(* CODESYS project CoDeSyS_library_v0.4.0.0.library
   LanguageModelAttribute: qualified-access-only
   Author: Razumovskii
   Version: 0.4.0.0
   Description: Standart library for main typical devices
   Title: mt
   Company: MechaTronics

Project tree, tasks and I/O mapping:
  libraries: Standard, 3.5.18.0 (System); Util, 3.5.19.0 (System); CAA File, 3.5.19.0 (CAA Technical Workgroup); CmpApp, 3.5.17.0 (System); SysTypes Interfaces, * (System)
  global variables sys
  System/
    program pou99_End [ST]: sysLoadZero, sysDevListReset, sysDevListCheck
    Library UDTs/
      data type udtDTL
      data type udtTimer
      data type timerSec
      data type timerRtc
      data type udtCMD
      data type timerCnt
      data type udtDevAnalog
      data type udtState
      data type udtDevDiscrete
      function devAtoD [ST]
      function devDtoA [ST]
      data type udtNetDataDiscrete
      data type udtNetDataAnalog
      data type uniSwap
    Library Methods/
      function GetLibVersion [ST]
      function block DrvBase [ST]: scale, conv, alm, almS, ot, exe, inc, blink, switch
      function block DrvTimer [ST]: sec, cnt, rtc
      function mbSwap [ST]
    program pou00_Start [ST]: pulse, clock, dtl, pulseOne
    Library Lists/
      data type listDev
      data type listRange
      data type listDevLoad
    function block DrvRetain [ST]: custom, system
  Drivers/
    Devices/
      02. Discrete Output/
        data type cfgDO
        data type cfgDOA
        function block DrvDO [ST]: s12_state, s15_globalData, s00_globalCommands, s05_exe, s09_options, s18_netData
        data type udtCfgDO
        function block DrvDOA [ST]: s12_state, s00_globalCommands, s01_externalCommand, s05_exe, s06_delays, s16_timers, s15_globalData, s07_turnON, s08_turnOFF, s09_options
      06. Valve Discrete/
        data type cfgV
        data type stateV
        function block DrvV [ST]: s00_globalCommands, s01_externalCommand, s04_alarmsRaw, s05_exe, s06_delays, s07_turnON, s08_turnOFF, s09_options, s10_alarms, s11_reset, s12_state, s14_opTime, s15_globalData, s16_timers, s17_hmi, s20_test, s18_netData
        data type udtCfgV
        data type udtAlarmV
        function block SubCalibration [ST]
      01. Discrete Input/
        data type cfgDI
        function block DrvDI [ST]: s00_globalCommands, s12_state, s02_workMode, s03_filter, s05_exe, s16_timers, s15_globalData, s09_options, s18_netData
        data type udtCfgDI
      05. Motor Direct/
        data type cfgM
        data type stateM
        function block DrvM [ST]: s16_timers, s15_globalData, s12_state, s00_globalCommands, s06_delays, s05_exe, s01_externalCommand, s09_options, s08_turnOFF, s07_turnON, s11_reset, s04_alarmsRaw, s10_alarms, s17_hmi, s14_opTime, s20_test, s18_netData
        data type udtCfgM
        data type udtAlarmM
      04. Analog Output/
        SlowMode/
          function block SubFilter [ST]
          function block SubSlow [ST]
          data type udtCfgSlow
          data type cfgSlow
        data type udtCfgAO
        data type cfgAO
        function block DrvAO [ST]: s12_state, s17_hmi, s15_globalData, s00_globalCommands, s01_externalCommand, s05_exe, s09_options, s18_netData
        data type stateAO
        function block DrvAO_MV210 [ST]: s12_state, s17_hmi, s15_globalData, s00_globalCommands, s01_externalCommand, s05_exe, s09_options, s04_alarmsRaw, s11_reset, s18_netData
        MV210/
          data type udtAO_MV210_502
          data type udtAlarmAO_MV210
          data type stateAO_MV210
      03. Analog Input/
        data type listAISp
        data type cfgAI
        data type stateAI
        data type udtAlarmAI
        data type udtCfgAI
        function block DrvAI [ST]: s07_turnON, s17_hmi, s04_alarmsRaw, s00_globalCommands, s10_alarms, s11_reset, s16_timers, s15_globalData, s02_workMode, s03_filter, s05_exe, s06_delays, s08_turnOFF, s09_options, s12_state, s18_netData
        function block DrvAI_MV210 [ST]: s07_turnON, s17_hmi, s04_alarmsRaw, s00_globalCommands, s10_alarms, s11_reset, s16_timers, s15_globalData, s02_workMode, s03_filter, s05_exe, s06_delays, s08_turnOFF, s09_options, s12_state, s18_netData
        MV210/
          data type udtAI_MV210_101
          data type udtAlarmAI_MV210
          data type stateAI_MV210
      20. PID/
        data type udtCfgPID
        data type cfgPID
        function block DrvPID [ST]: s07_turnON, s06_delays, s05_exe, s03_filter, s00_globalCommands, s09_options, s11_reset, s12_state, s15_globalData, s17_hmi, s13_commands
        data type statePID
        data type udtAlarmPID
      10. Flowmeter/
        function block DrvFlow [ST]: s00_globalCommands, s05_exe, s09_options, s11_reset, s12_state, s15_globalData, s16_timers, s17_hmi, s02_workMode, s03_filter, s18_netData
        data type udtCfgFlow
        data type cfgFlow
        data type stateFlow
    Special/
      function block DrvStatistics [ST]: calcD, addValue, reset, resetList, calcA, calcMulti
      data type listStatistic
      data type cfgStatistic
*)

// System/Library UDTs/udtDTL
TYPE udtDTL :
STRUCT
	//Data Time List
		year			:UINT;
		month			:UINT;
		day				:UINT;
		hour			:UINT;
		minute			:UINT;
		second			:UINT;
		millisecond		:UINT;
		weekDay			:WEEKDAY;
END_STRUCT
END_TYPE

// System/Library UDTs/udtTimer
TYPE udtTimer :
STRUCT
	//configuration word for Timers
		start		:BOOL;			// 0:	starting command
		Q			:BOOL;			// 1:	Quit
		pause		:BOOL;			// 2:	Pause
		reset		:BOOL;			// 3:	reset actual point to zero
		SFC			:BOOL;			// 4:	signal front control
		//you add more configuration bits for the project, if necessary, but not more than 16
END_STRUCT
END_TYPE

// System/Library UDTs/timerSec
TYPE timerSec :
STRUCT
	//control struct for a Timer Second
		cmd			:udtTimer;		//command word
		sp			:INT := 2;		//set point
		ap			:INT;			//actual point	
END_STRUCT
END_TYPE

// System/Library UDTs/timerRtc
TYPE timerRtc :
STRUCT
	//control struct for a Timer High Accucary
		cmd			:udtTimer;		//command word
		sp			:REAL := 2.000;	//set point as second
		ap			:REAL;			//actual point	
		RTC			:UDINT;			//real time stamp
		delta		:UDINT;			//delta time control
		percent		:REAL;			//progress 0..100%
END_STRUCT
END_TYPE

// System/Library UDTs/udtCMD
TYPE udtCMD :
STRUCT
	//standart control word
		startA	 		:BOOL;		// 0:	command for automatic control
		startM	 		:BOOL;		// 1:	command for manual control
		manual			:BOOL;		// 2:	mode of control (0 - automatic, 1 - manual (user or HMI))
		lock			:BOOL;		// 3:	technological lock
		force			:BOOL;		// 4:	forced control in manual mode
		service			:BOOL;		// 5:	activate service mode
		local			:BOOL;		// 6: 	activate local mode (0 - controlled by PLC, 1 - controlled by local keys)
		reset			:BOOL;		// 7:	resetting of device
		alarm			:BOOL;		// 8:	the device is in the alarm
		resetOT			:BOOL;		// 9:	reset opreational time
		direction		:BOOL;		// 10:	direction of moving
		lowSpeed		:BOOL;		// 11:	low speed mode
		test			:BOOL;		// 12:	test run for once		
		call			:BOOL;		// 13:	call device (0 - don't call, 1 - call)
		//you add more configuration bits for the project, if necessary, but not more than 15
END_STRUCT
END_TYPE

// Drivers/Devices/01. Discrete Input/cfgDI
TYPE cfgDI :
STRUCT
	cfg					:udtCfgDI;	// HMI 0:	configuration word
	//SP and another settings for Discrete Inputs
		spTOn			:REAL := 0.2;	// HMI 1:	SP Time chatter filter starting, seconds
		spTOff			:REAL := 0.2;	// HMI 2:	SP Time chatter filter before stoping, seconds
END_STRUCT
END_TYPE

//History log:
//2023.01.10
//	1) data type 'bit' -> 'bool'
//	2) delete memory optimisation

// Drivers/Devices/02. Discrete Output/cfgDO
TYPE cfgDO :
STRUCT
	cfg					:udtCfgDO;	// HMI 0:	configuration word
END_STRUCT
END_TYPE

// Drivers/Devices/02. Discrete Output/cfgDOA
TYPE cfgDOA :
STRUCT
	cfg					:udtCfgDO;	// HMI 0:	configuration word
	//SP and another settings for Discrete Outputs
		spT				:REAL;			// HMI 1:	SP Time for impulse or PWM mode
		spM				:REAL;			// HMI 3:	SP % for PWM mode in manual mode
		spMin			:REAL := 10;	// HMI 5:	SP minimum value for switch on
		spMax			:REAL := 90;	// HMI 7:	SP value, while not switch off
END_STRUCT
END_TYPE

// Drivers/Devices/05. Motor Direct/cfgM
TYPE cfgM :
STRUCT
	cfg					:udtCfgM;		// HMI 0:	configuration word
	//SP and another settings for Motors
		spTDelayOn		:INT;			// HMI 1:	SP Time delay before starting, seconds
		spTDelayOff		:INT;			// HMI 2:	SP Time delay before stoping, seconds
		spTOn			:INT := 2;		// HMI 3:	SP Time feedback control during start, seconds
		spTOff			:INT := 2;		// HMI 4:	SP Time feedback control during stop, seconds
		spTest			:INT := 3;		// HMI 5:	SP Time for running test
		opTime			:REAL;			// HMI 6:	Operation time, hours		
		opTimeLimit		:REAL;			// HMI 7:	Limit for operation time, hours	
		ID				:INT;			// HMI 5:	ID for SCADA
END_STRUCT
END_TYPE

//History log:
//2023.01.11
//	1) data type 'bit' -> 'bool'
//2023.01.18
//	1) delete service interval

// Drivers/Devices/05. Motor Direct/stateM
TYPE stateM :
STRUCT
	state				:udtState;			// HMI 0:	universal state word
	alarm				:udtalarmM;			// HMI 1:	alarm word for Motors
	signalQF			:BOOL;
	signalKM			:BOOL;
	//specified condition for Motors	
		status			:INT;				// HMI 2:	status code for HMI
		(*
			0 - Successfully stopped
			1 - Successfully started
			2 - In the process of stopping
			3 - In the process of starting
			4 - Service maintance
			5 - alarm "No Ready"
			6 - alarm when stopping / now ON
			7 - alarm when starting / now OFF
			8 - alarm TS
			9 - alarm SF
			10 - alarm communication
			11 - External alarm
			99 - emergency stop
			
			if any alarm, than device will try to stop
		*)
END_STRUCT
END_TYPE

//History log:
//2023.01.11
//	1) data type 'bit' -> 'bool'

// System/Library UDTs/timerCnt
TYPE timerCnt :
STRUCT
	//control struct for a Timer Millisecond or counting
		cmd			:udtTimer;		//command word
		sp			:REAL := 2.0;	//set point
		ap			:REAL;			//actual point
		one			:REAL := 0.1;	//impulse weight
		percent		:REAL;			//progress 0..100%
		PT			:R_TRIG;		//control of a positive signal front
END_STRUCT
END_TYPE

// System/Library Lists/listDev
TYPE listDev :
STRUCT
	//general types
		drvDI			:BOOL;		// 0:	any discrete input in *** mode or state
		drvDO			:BOOL;		// 1:	any discrete optput in *** mode or state
		drvAI			:BOOL;		// 2:	any analog input in *** mode or state
		drvAO			:BOOL;		// 3:	any analog ouput in *** mode or state
		drvM			:BOOL;		// 4:	any device type "M" in *** mode or state
		drvV			:BOOL;		// 5:	any device type "V" in *** mode or state
		drvAxis			:BOOL;		// 6:	any axis in *** mode or state
		Logick			:BOOL;		// 7:	any logical block in *** mode or state
		Unknown			:BOOL;		// 8:	something input/output or device in *** mode or state
		drvPID			:BOOL;		// 9:	any PID
		drvFlow			:BOOL;		// 10:	any flowmeter in *** mode or state
		drvCam			:BOOL;		// 11:	any camera in *** mode or state
		drvDOA			:BOOL;		// 12:	any DO with PWM in *** mode or state
		drvMR			:BOOL;		// 13:	any device type "MR" in *** mode or state	
		drvVFDsvt320	:BOOL;		// 14:	any VFD SVT320 in *** mode or state	
		
END_STRUCT
END_TYPE

// Drivers/Devices/06. Valve Discrete/cfgV
TYPE cfgV :
STRUCT
	cfg					:udtCfgV;		// HMI 0:	configuration word
	//SP and another settings for Valves
		spTDelayOn		:INT;			// HMI 1:	SP Time delay before starting, seconds
		spTDelayOff		:INT;			// HMI 2:	SP Time delay before stoping, seconds
		spTOn			:INT := 10;		// HMI 3:	SP Time feedback control during start, seconds
		spTOff			:INT := 10;		// HMI 4:	SP Time feedback control during stop, seconds
		spTest			:INT := 3;		// HMI 5:	SP Time for running test
		opTime			:REAL;			// HMI 6:	Operation time, hours		
		opTimeLimit		:REAL;			// HMI 7:	Limit for operation time, hours	
		ID				:INT;			// HMI 5:	ID for SCADA


END_STRUCT
END_TYPE

//History log:
//2023.01.13
//	1) data type 'bit' -> 'bool'
//	2) add TS, SF, SRV, Ext configurations
//	3) add SP_T_KM, fixed default SP time SP_T_ON/OFF '2 -> 10'

// Drivers/Devices/06. Valve Discrete/stateV
TYPE stateV :
STRUCT
	state				:udtState;			// HMI 0:	universal state word
	alarm				:udtalarmV;			// HMI 1:	alarm word for Valves
	signalQF			:BOOL;
	signalKM			:BOOL;
	signalOpen			:BOOL;
	signalClose			:BOOL;
	//specified condition for Valves
		status			:INT;					// HMI 2:	status code for HMI
		(*
			0 - Successfully stopped
			1 - Successfully started
			2 - In the process of stopping
			3 - In the process of starting
			4 - Service maintance
			5 - alarm "No Ready"
			6 - alarm when opening / now ON
			7 - alarm when closing / now OFF
			8 - alarm TS
			9 - alarm SF
			10 - alarm communication
			11 - External alarm
			12 - alarm while opening / now close
			13 - alarm while opening / now no FB
			14 - alarm while closing / now open
			15 - alarm while closing / now no FB
			99 - emergency stop
			
			if any alarm, than device will try to stop
		*)
END_STRUCT
END_TYPE

//History log:
//2023.01.11
//	1) data type 'bit' -> 'bool'

// System/Library UDTs/udtDevAnalog
TYPE udtDevAnalog :
STRUCT
	REQ				:BOOL;			//request for start device
	READY			:BOOL;			//device ready ready to control
	BUSY			:BOOL;			//device in start/stop process
	DONE			:BOOL;			//device succesfully started
	ALM				:BOOL;			//device has critical alarm
	STATUS			:INT;
	SP				:REAL;			//setpoint for device
	AP				:REAL;			//actual point (position, speed, etc)
END_STRUCT
END_TYPE

// Drivers/Devices/02. Discrete Output/udtCfgDO
TYPE udtCfgDO :
STRUCT
	//configuration struct for Discrete Outputs
		useSim			:BOOL;			// PLC 0:	0 - Normal mode of operation, 		1 - Simulation mode
		useNoEmrg		:BOOL;			// HMI 1:	0 - Use emergency signal,			1 - Ignore emergency signal
		useExt			:BOOL := TRUE;	// HMI 2:	0 - Use internal command,			1 - Use external command
		useNC			:BOOL;			// HMI 3:	0 - Normal Open signal, 			1 - Normal Close signal
		useImpulse		:BOOL;			// HMI 4:	0 - Permanent mode of operation, 	1 - Impulse mode of operation
		usePWM			:BOOL;			// HMI 5:	0 - Constant signal,				1 - PWM signal
		//you may add more configuration bits for the project, if necessary, but not more than 15
END_STRUCT
END_TYPE

// Drivers/Devices/05. Motor Direct/udtCfgM
TYPE udtCfgM :
STRUCT
	//configuration word for Motors
		useSim			:BOOL;			// HMI 0:	0 - Normal mode of operation,	1 - Simulation mode
		useNoEmrg		:BOOL;			// HMI 1:	0 - Use emergency signal,		1 - Ignore emergency signal
		useExt			:BOOL := FALSE;	// HMI 2:	0 - Use internal command,		1 - Use external command
		useQF			:BOOL := TRUE;	// HMI 3:	Feedback control "Ready"
		useKM			:BOOL := TRUE;	// HMI 4:	Feedback control "In work"
		useOT			:BOOL := TRUE;	// HMI 5:	Control operation time
		//you may add more configuration bits for the project, if necessary, but not more than 15
END_STRUCT
END_TYPE

// Drivers/Devices/01. Discrete Input/udtCfgDI
TYPE udtCfgDI :
STRUCT
	//configuration struct for Discrete Inputs
		useSim			:BOOL;			// PLC 0:	0 - Normal mode of operation, 	1 - Simulation mode
		useNoEmrg		:BOOL;			// HMI 1:	0 - Use emergency signal,		1 - Ignore emergency signal
		useNC			:BOOL;			// HMI 2:	0 - Normal Open signal, 		1 - Normal Close signal
		useFilter		:BOOL;			// HMI 3:	0 - Not use filter,				1 - Use chatter filter
		//you may add more configuration bits for the project, if necessary, but not more than 15
END_STRUCT
END_TYPE

// System/Library UDTs/udtState
TYPE udtState :
STRUCT
	//unviversal condition word for any devices
		call			:BOOL;		// 0:	call device (0 - don't call, 1 - call)
		enable			:BOOL;		// 1:	device enabled
		alarm			:BOOL;		// 2:	device in something alarm
		ready			:BOOL;		// 3:	device ready to start		
		busy			:BOOL;		// 4:	device busy and working now
		done			:BOOL;		// 5:	device finished task
		posOk			:BOOL;		// 6:	position/speed reached or run now
		local			:BOOL;		// 7:	device in local mode
		service			:BOOL;		// 8:	device in service mode
		warningOT		:BOOL;		// 9:	warning "Service maintenance is required, the interservice interval is exceeded"
		//you may add more configuration bits for the project, if necessary, but not more than 15
END_STRUCT
END_TYPE

// Drivers/Devices/05. Motor Direct/udtAlarmM
TYPE udtalarmM :
STRUCT
	//alarm word for Motors
		almQF			:BOOL;		// 0:	alarm "No Ready" 
		almStart		:BOOL;		// 1:	alarm "No In Work when starting"
		almStop			:BOOL;		// 2:	alarm "In Work when stopping"
		almTS			:BOOL;		// 3:	alarm "No TS"
		almSF			:BOOL;		// 4:	alarm "No Safety signal"
		almExt			:BOOL;		// 5:	alarm "External alarm"
		almLink			:BOOL;		// 6:	alarm communication
		almES			:BOOL;		// 7:	alarm "emergency Stop"
		//you may add more configuration bits for the project, if necessary, but not more than 15
END_STRUCT
END_TYPE

// Drivers/Devices/06. Valve Discrete/udtCfgV
TYPE udtCfgV :
STRUCT
	//configuration struct for Valves
		//configuration word for Valves
		useSim			:BOOL;			// HMI 0:	0 - Normal mode of operation,	1 - Simulation mode
		useNoEmrg		:BOOL;			// HMI 1:	0 - Use emergency signal,		1 - Ignore emergency signal
		useExt			:BOOL := FALSE;	// HMI 2:	0 - Use internal command,		1 - Use external command
		useQF			:BOOL := TRUE;	// HMI 3:	Feedback control "Ready"
		usefbOpen		:BOOL := TRUE;	// HMI 4:	Feedback control "Valve Opened"
		usefbClose		:BOOL := TRUE;	// HMI 5:	Feedback control "Valve Closed"
		useNetwork		:BOOL := FALSE;	// HMI 6:	Use network connection
		useOT			:BOOL := TRUE;	// HMI 7:	Control operation time
		useSignal 		:BOOL := TRUE;	// HMI 8:	Use external REQ
		useCWF			:BOOL := TRUE;	// HMI 9:	Close While Fault
		useAir			:BOOL;			// HMI 10:	Work mode for air valves
		useDuo			:BOOL;			// HMI 11:	Work mode for CW/CCW
		useOnce			:BOOL;			// HMI 12:	Work mode without open/close feedback control after finishing movement
END_STRUCT
END_TYPE

// Drivers/Devices/06. Valve Discrete/udtAlarmV
TYPE udtalarmV :
STRUCT
	//alarm word for Valves
		almQF			:BOOL;		// 0:	alarm "No Ready" 
		almOpen			:BOOL;		// 1:	alarm while opening
		almClose		:BOOL;		// 2:	alarm while closing
		almTS			:BOOL;		// 3:	alarm "No TS"
		almDuo 			:BOOL;		// 4:	alarm duo signals fbOpen and fbClose at once
		almExt			:BOOL;		// 5:	alarm "External alarm"
		almLink			:BOOL;		// 6:	alarm communication
		almES			:BOOL;		// 7:	alarm "emergency Stop"
		//you may add more configuration bits for the project, if necessary, but not more than 15
END_STRUCT
END_TYPE

// Drivers/Devices/03. Analog Input/listAISp
TYPE listAISp :
STRUCT
	HH			:REAL := 90;
	H			:REAL := 75;
	L			:REAL := 25;
	LL			:REAL := 10;
	SC			:REAL := 105;
	NC			:REAL := -5;
END_STRUCT
END_TYPE

// System/Library Lists/listRange
TYPE listrange :
STRUCT
	minIn		:REAL := 0;
	maxIn		:REAL := 100;
	minOut		:REAL := 0;
	maxOut		:REAL := 100;
END_STRUCT
END_TYPE

// Drivers/Devices/03. Analog Input/cfgAI
TYPE cfgAI :
STRUCT
	//configuration struct for Analog Inputs
		cfg				:udtCfgAI;		// HMI 0:	configuration word
		inputType		:INT := 1;		// HMI 1:	Input type: 0 = 0..20, 1 = 4..20, 2 = 0..10, 3 = Pt100, 4 = Pt1000
		valueType		:INT := 0;		// HMI 2:	value type: 0 = %, 1 = Hz, 2 = l/h, etc
		filterType		:INT := 1;		// HMI 3:	Execution clock for filter: 0 = every cycle of PLC, 1 = 0.1s, 2 = 1s
		filterLim		:INT := 100;	// HMI 4:	value of records in filter buffer
		range			:listRange;		// HMI 5:	Singal scale range
		calibration		:REAL;			// HMI 13:	Static correction
		multiplier		:REAL := 1;		// HMI 15:	Multiple correction
		sp				:listAIsp;		// HMI 17:	SP for limits
		spT				:ARRAY [0..3] OF INT;// HMI 26:	SP timers for limits
		ID				:INT;			// HMI 5:	ID for SCADA
		// HMI x - x is word number in shift address by start address
END_STRUCT
END_TYPE

// Drivers/Devices/03. Analog Input/stateAI
TYPE stateAI :
STRUCT
	//condition for Analog Inputs
		state		:udtState;			// PLC 0:	condition word
		alarm		:udtalarmAI;		// HMI 1:	alarm word
		status		:INT;				// HMI 2:	status code for HMI
		result		:REAL;				// HMI 3:	signal from analog input in sensor range
		signal		:REAL;				// HMI 5:	signal from analog input in phisycal range
		(*	status:
			0 - disable
			1 - result > L and result < H
			2 - result < L and result > LL
			3 - result > H and result < HH
			4 - alarm "ST"
			5 - alarm "NC"
			6 - alarm LL
			7 - alarm HH
			
			if any alarm, than HMI will send message
		*)
END_STRUCT
END_TYPE

// Drivers/Devices/03. Analog Input/udtAlarmAI
TYPE udtalarmAI :
STRUCT
	//alarm word for Analog Inputs
		almST		:BOOL;		// 0:	alarm "No Ready" 
		almHH		:BOOL;		// 1:	alarm "High alarm level"
		almH		:BOOL;		// 2:	warning "High work level"
		almL		:BOOL;		// 3:	warning "Low work level"
		almLL		:BOOL;		// 4:	alarm "Low alarm level"
		almNC		:BOOL;		// 5:	alarm "No connect"
		almSC		:BOOL;		// 6:	alarm "Overload"
		//you add more configuration bits for the project, if necessary, but not more than 16
END_STRUCT
END_TYPE

// Drivers/Devices/03. Analog Input/udtCfgAI
TYPE udtCfgAI :
STRUCT
	//configuration word for Analog Inputs
		useSim			:BOOL;			// PLC 0:	0 - Normal mode of operation, 	1 - Simulation mode
		useNoEmrg		:BOOL;			// PLC 1:	0 - Use emergency signal,		1 - Ignore emergency signal
		useEnable		:BOOL := TRUE;
		useRTD			:BOOL := FALSE;	// HMI 2:	Use mode RTD/TC scaling
		useFilter		:BOOL := TRUE;	// HMI 3:	Use filter
		useLight		:BOOL;			// HMI 4:	Lighting status for screen indication
		useLow			:BOOL := TRUE;	// PLC 5:	Enable low level alarms
		useHigh			:BOOL := TRUE;	// PLC 6:	Enable high level alarms
		useSC			:BOOL;			// HMI 7:	use control wire break
		useAutoreset	:BOOL;			// HMI 8:	use auto reset for HH and LL alarms
		useCompact		:BOOL;			// HMI 9:	use compact form with ready-to-work input value
		//you add more configuration bits for the project, if necessary, but not more than 16
END_STRUCT
END_TYPE

// System/Library UDTs/udtDevDiscrete
TYPE udtDevDiscrete :
STRUCT
	REQ				:BOOL;			//request for start device
	READY			:BOOL;			//device ready ready to control
	BUSY			:BOOL;			//device in start/stop process
	DONE			:BOOL;			//device succesfully started
	ALM				:BOOL;			//device has critical alarm
	STATUS			:INT;
END_STRUCT
END_TYPE

// Drivers/Devices/04. Analog Output/udtCfgAO
TYPE udtCfgAO :
STRUCT
	//configuration word for Analog Outputs
		useSim			:BOOL;			// PLC 0:	0 - Normal mode of operation, 	1 - Simulation mode
		useNoEmrg		:BOOL;			// HMI 1:	0 - Use emergency signal,		1 - Ignore emergency signal
		useExt			:BOOL;			// HMI 2:	0 - Use internal command,			1 - Use external command
		useLight		:BOOL;			// HMI 3:	Lighting status for screen indication
		useSlow			:BOOL;			// HMI 4:	0 - normal mode, 				1 - slow mode
		//you add more configuration bits for the project, if necessary, but not more than 16
END_STRUCT
END_TYPE

// Drivers/Devices/04. Analog Output/cfgAO
TYPE cfgAO :
STRUCT
	//configuration struct for Analog Outputs
		cfg				:udtCfgAO;		// HMI 0:	configuration word
		outputType		:INT := 1;		// HMI 1:	Output type: 0 = 0..20, 1 = 4..20, 2 = 0..10, 3 = Pt100, 4 = Pt1000
		valueType		:INT := 0;		// HMI 2:	value type: 0 = %, 1 = Hz, 2 = l/h, etc
		range			:listrange;		// HMI 3:	Singal scale range
		spM				:REAL;			// HMI 10:	SP in manual mode
		slowCfg			:cfgSlow;		// HMI 11:
		ID				:INT;			// HMI 5:	ID for SCADA		
END_STRUCT
END_TYPE

// Drivers/Devices/04. Analog Output/stateAO
TYPE stateAO :
STRUCT
	//condition for Analog Inputs
		state		:udtState;			// HMI 0:	condition word
		status		:INT;				// HMI 1:	status code for HMI
		result		:REAL;				// HMI 2:	command for analog output in device range
		signal		:REAL;				// HMI 4:	command for analog output in phisycal range
		slowState	:udtState;			// HMI 5:	Slow mode state
		(*	status:
			0 - disable
			1 - activate
			
			if any alarm, than HMI will send message
		*)
END_STRUCT
END_TYPE

// Drivers/Devices/10. Flowmeter/udtCfgFlow
TYPE udtCfgFlow :
STRUCT
	//configuration word for Analog Inputs
		useSim		:BOOL;			// PLC 0:	0 - Normal mode of operation, 	1 - Simulation mode
		useNoEmrg	:BOOL;			// PLC 1:	0 - Use emergency signal,		1 - Ignore emergency signal
		usePOU		:BOOL := TRUE;  // HMI 2:	Call FE in special POU with fixed time
		useFilter	:BOOL := TRUE;	// HMI 3:	Use filter
		useLight	:BOOL;			// HMI 4:	Lighting status for screen indication
		useDI		:BOOL := TRUE;	// HMI 5:	Use DI signal
		useFM		:BOOL;			// HMI 6:	Use weight control
		useFMAdd	:BOOL;			// HMI 7:	Use add weight control
		usePreSP	:BOOL := TRUE;	// HMI 8:	Use pre-SP  control
		useSP		:BOOL := TRUE;	// HMI 9:	Use SP control
		//you add more configuration bits for the project, if necessary, but not more than 16
END_STRUCT
END_TYPE

// Drivers/Devices/10. Flowmeter/cfgFlow
TYPE cfgFlow :
STRUCT
	//configuration struct for FlowMeter
		cfg				:udtCfgFlow;	// HMI 0:	configuration word
		weight			:REAL := 0.1;	// HMI 1:	Weight for 1 impulse
		sizeWeight		:INT := 0;		// HMI 3:	Wieght of control unit - ml, l, m3
		sizeTime		:INT;			// HMI 5:	Speed of flow size: 0 - hour, 1 - minute, 2 - second
		filterLim		:INT := 10;		// HMI 6:	Filter limit for summ values, max = 100
		filterType		:INT;			// HMI 7:	Execution clock for filter: 0 = every cycle of PLC, 1 = 0.1s, 2 = 1s
		clock			:INT := 2;		// HMI 8:	Cycle time for POU mode, ms
		seans			:REAL;			// HMI 9:	Last seans data
		spPre			:REAL;			// HMI 11:	Presetpoint for one seans control
		sp				:REAL := 1;		// HMI 13:	Setpoint for one seans control
		db				:REAL := 0.1;	// HMI 15:	Deadband for setpoint
END_STRUCT
END_TYPE

// Drivers/Devices/10. Flowmeter/stateFlow
TYPE stateFlow :
STRUCT
	//condition for Analog Inputs
		state		:udtState;			// HMI 0:	condition word
		status		:INT;				// HMI 1:	status code for HMI
		result		:REAL;				// HMI 2:	Actual flow speed
		ap			:REAL;				// HMI 4:	Actual flow value
		lastAp		:REAL;				// HMI 6:	Last flow value
		(*
			0 - disable
			1 - result > L and result < H
			2 - result < L and result > LL
			3 - result > H and result < HH
			4 - alarm "ST"
			5 - alarm "NC"
			6 - alarm LL
			7 - alarm HH
			
			if any alarm, than HMI will send message
		*)
END_STRUCT
END_TYPE

// Drivers/Devices/04. Analog Output/SlowMode/udtCfgSlow
TYPE udtCfgSlow :
STRUCT
	//configuration struct for sub driver Slow
		//configuration word for Valves
		enable			:BOOL;			// HMI 0:	Enable algorythm
		useUp			:BOOL;			// HMI 1:	use slow mode for up value
		useDown			:BOOL;			// HMI 2:	use slow mode for down value
		useForceUp		:BOOL;			// HMI 3:	use force mode for first up
		useForceDown	:BOOL;			// HMI 4:	use force mode for last down
END_STRUCT
END_TYPE

// Drivers/Devices/04. Analog Output/SlowMode/cfgSlow
TYPE cfgSlow :
STRUCT
	cfg					:udtCfgSlow;	// HMI 0:	configuration word
	//SP and another settings for sub driver Slow
		spMin			:REAL;
		spMax			:REAL;
		spStepUp		:REAL;
		spStepDown		:REAL;
		spTUp			:REAL;
		spTDown			:REAL;
END_STRUCT
END_TYPE

// System/Library Lists/listDevLoad
TYPE listDevLoad :
STRUCT
	//general types
		drvDI			:INT;		// 0:	any discrete input in *** mode or state
		drvDO			:INT;		// 1:	any discrete optput in *** mode or state
		drvAI			:INT;		// 2:	any analog input in *** mode or state
		drvAO			:INT;		// 3:	any analog ouput in *** mode or state
		drvM			:INT;		// 4:	any device type "M" in *** mode or state
		drvV			:INT;		// 5:	any device type "V" in *** mode or state
		drvAxis			:INT;		// 6:	any axis in *** mode or state
		Logick			:INT;		// 7:	any logical block in *** mode or state
		Unknown			:INT;		// 8:	something input/output or device in *** mode or state
		drvPID			:INT;		// 9:	any PID
		drvFlow			:INT;		// 10:	any flowmeter in *** mode or state
		drvCam			:INT;		// 11:	any camera in *** mode or state
		drvDOA			:INT;		// 12:	any DO with PWM in *** mode or state
		drvMR			:INT;		// 13:	any device type "MR" in *** mode or state	
		drvVFDsvt320	:INT;		// 14:	any VFD SVT320 in *** mode or state	
END_STRUCT
END_TYPE

// Drivers/Devices/20. PID/udtCfgPID
TYPE udtCfgPID :
STRUCT
	//configuration word for PID
		useSim			:BOOL;			// HMI 0:	0 - Normal mode of operation,	1 - Simulation mode
		useNoEmrg		:BOOL;			// HMI 1:	0 - Use emergency signal,		1 - Ignore emergency signal
		useScaleIn		:BOOL;
		useScaleOut		:BOOL;
		useCorrectionIn	:BOOL;
		useCorrectionOut:BOOL;
		useDB			:BOOL;
END_STRUCT
END_TYPE

// Drivers/Devices/20. PID/cfgPID
TYPE cfgPID :
STRUCT
	//configuration struct for PID
		cfg				:udtCfgPID;		// HMI 0:	configuration word
		spA				:REAL := 1.0;
		spM				:REAL := 1.0;
		spDB			:REAL := 0.1;
		spResult		:REAL;
		rangeIn			:listRange;		// HMI 5:	Singal input scale range
		rangeOut		:listRange;		// HMI 5:	Singal output scale range
		spKP			:REAL := 1.0;
		spTi			:REAL := 125.0;
		spTd			:REAL := 0.0;
		calibrationIn	:REAL;			// HMI 13:	Static correction
		multiplierIn	:REAL := 1;		// HMI 15:	Multiple correction
		calibrationOut	:REAL;			// HMI 13:	Static correction
		multiplierOut	:REAL := 1;		// HMI 15:	Multiple correction
		typeInput		:INT := 0;
		typeOutput		:INT := 0;
		ID				:INT;			// HMI 30:	ID for SCADA
		name			:ARRAY [0..9] OF BYTE; // HMI 31:	Name
		ADDR			:INT;			// PLC xx:	address of inputs
END_STRUCT
END_TYPE

// Drivers/Devices/20. PID/statePID
TYPE statePID :
STRUCT
	state				:udtState;			// HMI 0:	universal state word
	alarm				:udtAlarmPID;		// HMI 1:	alarm word for Motors
	signalPID			:REAL;
	resultPID			:REAL;
END_STRUCT
END_TYPE

// Drivers/Devices/20. PID/udtAlarmPID
TYPE udtAlarmPID :
STRUCT
	//alarm word for PID
		almLimits		:BOOL;		// 0:	TRUE: Y has exceeded the given limits Y_MIN, Y_MAX and is limited to these values
		almOveFlow		:BOOL;		// 1:	Overflow in integral part
END_STRUCT
END_TYPE

// Drivers/Devices/03. Analog Input/MV210/udtAI_MV210_101
TYPE udtAI_MV210_101 :
STRUCT
	signal			:REAL;	//input value
	cycleTime		:UINT;
	errorCode		:USINT;
END_STRUCT
END_TYPE

// Drivers/Devices/04. Analog Output/MV210/udtAO_MV210_502
TYPE udtAO_MV210_502 :
STRUCT
	signal			:UINT;	//output checkdata
	value			:UINT;	//output setpoint
	errorCode		:USINT;
END_STRUCT
END_TYPE

// Drivers/Devices/04. Analog Output/MV210/udtAlarmAO_MV210
TYPE udtAlarmAO_MV210 :
STRUCT
	//alarm word for Analog Inputs
		NO_DAC_CONNECTION		:BOOL;//			1	Нет связи с ЦАП
		NO_LOAD					:BOOL;//			2	Отсутствие нагрузки
		DAC_OVERHEAT			:BOOL;//			3	Перегрев ЦАП
		CRC_ERROR				:BOOL;//			4	Ошибка CRC
		CHANNEL_DISABLED		:BOOL;//			5	Канал отключен
		SHORT_CIRCUIT			:BOOL;//			6	Короткое замыкание
		//you add more configuration bits for the project, if necessary, but not more than 16
END_STRUCT
END_TYPE

// Drivers/Devices/03. Analog Input/MV210/udtAlarmAI_MV210
TYPE udtAlarmAI_MV210 :
STRUCT
	//alarm word for Analog Inputs MV210
		almST		:BOOL;		// 0:	alarm "No Ready" 
		almHH		:BOOL;		// 1:	alarm "High alarm level"
		almH		:BOOL;		// 2:	warning "High work level"
		almL		:BOOL;		// 3:	warning "Low work level"
		almLL		:BOOL;		// 4:	alarm "Low alarm level"
		almNC		:BOOL;		// 5:	alarm "No connect"
		almSC		:BOOL;		// 6:	alarm "Overload"
		FIELDBUS_ERROR			:BOOL;//			241	Нет связи с модулем
		INCORRECT_VALUE			:BOOL;//			240	Заведомо неверное значение
		DATA_NOT_READY			:BOOL;//			246	Данные не готовы
		SENSOR_DISABLED			:BOOL;//			247	Датчик отключен
		TOO_HIGH_TEMP			:BOOL;//			248	Велика температура свободных концов ТП
		TOO_LOW_TEMP			:BOOL;//			249	Мала температура свободных концов ТП
		TOO_HIGH_VALUE			:BOOL;//			250	Значение велико
		TOO_LOW_VALUE			:BOOL;//			251	Значение мало
		SHORT_CIRCIUT			:BOOL;//			252	Короткое замыкание
		SENSOR_FAILED			:BOOL;//			253	Обрыв датчика
		NO_CONNECTION_TO_ADC	:BOOL;//			254	Нет связи с АЦП
		INCORRECT_CALIBRATION	:BOOL;//			255	Некорректная калибровка
		//you add more configuration bits for the project, if necessary, but not more than 16
END_STRUCT
END_TYPE

// Drivers/Devices/03. Analog Input/MV210/stateAI_MV210
TYPE stateAI_MV210 :
STRUCT
	//condition for Analog Inputs
		state		:udtState;			// PLC 0:	condition word
		alarm		:udtAlarmAI_MV210;
		status		:INT;				// HMI 2:	status code for HMI
		result		:REAL;				// HMI 3:	signal from analog input in sensor range
		signal		:REAL;				// HMI 5:	signal from analog input in phisycal range
		(*	status:
			0 - disable
			1 - result > L and result < H
			2 - result < L and result > LL
			3 - result > H and result < HH
			4 - alarm "ST"
			5 - alarm "NC"
			6 - alarm LL
			7 - alarm HH
			
			if any alarm, than HMI will send message
		*)
END_STRUCT
END_TYPE

// Drivers/Devices/04. Analog Output/MV210/stateAO_MV210
TYPE stateAO_MV210 :
STRUCT
	//condition for Analog Inputs
		state		:udtState;			// HMI 0:	condition word
		almMV210	:udtAlarmAO_MV210;
		status		:INT;				// HMI 1:	status code for HMI
		result		:REAL;				// HMI 2:	command for analog output in device range
		signal		:REAL;				// HMI 4:	command for analog output in phisycal range
		slowState	:udtState;			// HMI 5:	Slow mode state
		(*	status:
			0 - disable
			1 - activate
			
			if any alarm, than HMI will send message
		*)
END_STRUCT
END_TYPE

// Drivers/Special/listStatistic
TYPE listStatistic :
STRUCT
	seans			:REAL;
	lastSeans		:REAL;
	hour			:REAL;
	day				:REAL;
	week			:REAL;
	month			:REAL;
	year			:REAL;
	total			:REAL;
END_STRUCT
END_TYPE

// Drivers/Special/cfgStatistic
TYPE cfgStatistic :
STRUCT
	useDiscrete			:BOOL;
	useAnalog			:BOOL;
	useSkip				:BOOL;
	useClock			:BOOL;
	reset				:BOOL;
	resetWork			:BOOL;
	resetSkip			:BOOL;
	resetAll			:BOOL;
	weightD				:REAL := 0.01;
	weightA				:INT := 0;		//0 - hour, 1 - minutes, 2 - seconds
	weightClock			:REAL := 0.002;//cicle time in ms
	work				:listStatistic;
	skip				:listStatistic;
	all					:listStatistic;
END_STRUCT
END_TYPE

// System/Library UDTs/udtNetDataDiscrete
TYPE udtNetDataDiscrete :
STRUCT
	status					:INT;
	alarm					:WORD;
END_STRUCT
END_TYPE

// System/Library UDTs/udtNetDataAnalog
TYPE udtNetDataAnalog :
STRUCT
	status					:INT;
	alarm					:WORD;
	ap						:REAL;
END_STRUCT
END_TYPE

// System/Library UDTs/uniSwap
TYPE uniSwap :
UNION
	value		:DWORD;
	source		:ARRAY [0..1] OF WORD;
END_UNION
END_TYPE

// sys
{attribute 'qualified_only'}
VAR_GLOBAL
	//General management
		//Global controls
			allBlock				:BOOL;				//emergency stop
			allReset				:BOOL;				//reset all alarms
			allSim					:BOOL;				//Switch simulation mode for all devices
			allAuto					:BOOL;				//reset "CMD.manual" for all devices
			silence					:BOOL;				//Disable siren from HMI
			retainSave				:BOOL;				//Save data from Retain/PVL to file
			retainLoad				:BOOL;				//Read data to Retain/PVL from file
			loadZero				:BOOL;				//Load 0 to all buffers
		//Service tags
			alm						:listDev;			//alarms flags for devices
			man						:listDev;			//manual flags for devices
			sim						:listDev;			//Simulation flags for devices
			dataSave				:BOOL;
			dataLoad				:BOOL;
			DAT						:DATE_AND_TIME;					//System time
			DTL						:udtDTL;						//System time
			DTLnew					:udtDTL;						//System time
			DTLpulse				:udtDTL;						//System time
			upTime					:TIME;							//Work time after power on
			upTimeMs				:UDINT;							//Work time after power on as millisecond
		//Global data
			libVersion				:VERSION;			//Version code
			retainFileName 		:STRING := 'App1.ret';			//file name for Retain/PVL variables
		
		//Additional tags and constans
			second					:REAL := (1.0/3600.0);			//wight of 1 second in hour format
			dev						:INT;							//device counter for FOR
			alwsON					:BOOL := TRUE;					//always TRUE
			alwsOFF					:BOOL := FALSE;					//always FALSE
			startUp_Load			:BOOL;							//First load configuration after power on
				
		//Impulse tags
			pulse01s				:BOOL;							//global trigger 100 ms
			pulse1s					:BOOL;							//global trigger 1 second
			pulseMinute				:BOOL;							//global trigger 1 minute
			pulseHour				:BOOL;							//global trigger 1 hour
			pulseDay				:BOOL;							//global trigger 1 day
			pulseMonth				:BOOL;							//global trigger 1 month
			pulseYear				:BOOL;							//global trigger 1 year
			
		//clock tags
			clock01s				:BOOL;							//global clock for 100 ms
			clock05s				:BOOL;							//global clock for 500 ms
			clock1s					:BOOL;							//global clock for 1 s
			
		//Buffer for drivers
			load					:listDevLoad;	//requestment device ID
			actual					:listDevLoad;	//loaded device ID
			
		//Global functional blocks
			timer					:DrvTimer;
			base					:DrvBase;
			retainControl			:DrvRetain;
			
		//Special variables for Drv
			aiMaxValueType			:INT := 3;
			aiMaxValueValue			:INT := 10;
			aiMaxValueFilter		:INT := 2;
			aoMaxValueType			:INT := 2;
			aoMaxValueValue			:INT := 5;
END_VAR

// System/pou99_End
PROGRAM pou99_End
VAR
END_VAR

//cleaning buffer of loaded devices
	sysLoadZero();

//manual signal processing
	IF sysDevListCheck(dev_list := sys.man) THEN
		sys.man.Unknown := TRUE;
	ELSE
		sys.man.Unknown := FALSE;
	END_IF;

//error signal processing
	IF sysDevListCheck(dev_list := sys.alm) THEN
		sys.alm.Unknown := TRUE;
	ELSE
		sys.alm.Unknown := FALSE;
	END_IF;
	
//simulation signal processing
	IF sysDevListCheck(dev_list := sys.sim) THEN
		sys.sim.Unknown := TRUE;
	ELSE
		sys.sim.Unknown := FALSE;
	END_IF;
	
//reset alarm processing
	IF sys.allreset THEN
		sysDevListreset(dev_list := sys.alm);
		sys.allreset := FALSE;
		sys.Silence := FALSE;
	END_IF;

//reset auto
	IF sys.allAuto THEN
		sysDevListreset(dev_list := sys.man);
		sys.allAuto := FALSE;
	END_IF

ACTION sysLoadZero:
//cleaning device buffer
IF sys.loadZero THEN
	sys.load.drvAI 			:= 0;
	sys.load.drvAO 			:= 0;
	sys.load.drvDI 			:= 0;
	sys.load.drvDO 			:= 0;
	sys.load.drvM 			:= 0;
	sys.load.drvV	 		:= 0;
	sys.load.drvMR 			:= 0;
	sys.load.drvAxis 		:= 0;
	sys.load.drvCam 		:= 0;
	sys.load.drvDOA 		:= 0;
	sys.load.drvPID 		:= 0;
	sys.load.drvVFDsvt320	:= 0;
	sys.loadZero 			:= FALSE;
END_IF
END_ACTION

METHOD sysDevListReset : BOOL
VAR_IN_OUT
	dev_list 				:listDev;
END_VAR
//reset all variables in dev_list
	dev_list.drvDI			:= FALSE;
	dev_list.drvDO			:= FALSE;
	dev_list.drvAI			:= FALSE;
	dev_list.drvAO			:= FALSE;
	dev_list.drvM			:= FALSE;
	dev_list.drvV			:= FALSE;
	dev_list.drvAxis		:= FALSE;
	dev_list.Logick			:= FALSE;
	dev_list.Unknown		:= FALSE;
	dev_list.drvPID			:= FALSE;
	dev_list.drvFlow		:= FALSE;
	dev_list.drvCam			:= FALSE;
	dev_list.drvDOA			:= FALSE;
	dev_list.drvMR			:= FALSE;
	dev_list.drvVFDsvt320	:= FALSE;
END_METHOD

METHOD sysDevListCheck : BOOL
VAR_INPUT
	dev_list 				:listDev;
END_VAR
//Check if any variables in dev_list is TRUE
	IF 
		   dev_list.drvDI
		OR dev_list.drvDO
		OR dev_list.drvAI
		OR dev_list.drvAO
		OR dev_list.drvM
		OR dev_list.drvV
		OR dev_list.drvAxis
		OR dev_list.Logick
		OR dev_list.drvPID
		OR dev_list.drvFlow
		OR dev_list.drvCam
		OR dev_list.drvDOA
		OR dev_list.drvMR
		OR dev_list.drvVFDsvt320
	THEN
		sysDevListCheck := TRUE;
	ELSE
		sysDevListCheck := FALSE;
	END_IF
END_METHOD

END_PROGRAM

// Drivers/Devices/03. Analog Input/DrvAI
FUNCTION_BLOCK DrvAI
VAR_INPUT
	signal			:REAL;			//Analog input signal from PLC
END_VAR	
VAR_IN_OUT
	CMD				:udtCMD;		//Non-retain structure with command word
	cfg				:cfgAI;			//Retain structure with settings
END_VAR
VAR_OUTPUT
	state			:stateAI;		//Non-retain structure with states information
	netData			:udtNetDataAnalog;	//Data for network communication via ModBus TCP/RTU
	result			:REAL;			//signal from sensor
END_VAR
VAR
	value			:REAL;			//tmp value for calculating 
	buffer			:REAL;			//tnp value for slow mode
	emergency		:BOOL;			//emergency signal
	cnt				:INT;			//internal counter
	PT				:ARRAY [0..1] OF R_TRIG;
	NT				:ARRAY [0..1] OF F_TRIG;
	clock			:ARRAY [0..3] OF timerRtc;
	Filter			:subFilter;
END_VAR

//ANALOG INPUT
//control of typical analog sensors
// - pressure
// - level
// - flowmeter
// - etc

s00_globalCommands();
IF NOT cfg.cfg.useCompact THEN
	//s01_externalCommand();
	s02_workMode();
	s03_filter();
	s04_alarmsRaw();
END_IF
s05_exe();
//s06_delays();
//s07_turnON();
//s08_turnOFF();
s09_options();
s10_alarms();
s11_reset();
s12_state();
//s13_commands();
//s14_opTime();
s15_globalData();
s16_timers();
s17_hmi();
s18_netData();
//s19_reserv();
//s20_test();

ACTION s07_turnON:

END_ACTION

ACTION s17_hmi:
//hmi data
	//input scaling
		state.signal := sys.base.scale(
			value := signal,
			inputType := cfg.inputType,
			range := cfg.range);
	//rotate input type
		cfg.inputType := sys.base.inc(
			rotate := cmd.test,
			value := cfg.inputType,
			maxValue := sys.aiMaxValueType);
	//rotate value type
		cfg.valueType := sys.base.inc(
			rotate := cmd.lowSpeed,
			value := cfg.valueType,
			maxValue := sys.aiMaxValueValue);
	//rotate filter type
		cfg.filterType := sys.base.inc(
			rotate := cmd.local,
			value := cfg.filterType,
			maxValue := sys.aiMaxValueFilter);
END_ACTION

ACTION s04_alarmsRaw:
//alarms raw
	
	//SC control
	IF cfg.cfg.useSC AND CMD.startA  THEN
		CASE cfg.inputType OF 
			0: 	//0..20 mA
				state.alarm.almSC := sys.base.almS(
					signal := state.signal > 21.0,
					reset := cmd.reset);
			1: 	//4..20 mA
				state.alarm.almSC := sys.base.almS(
					signal := state.signal > 21.0,
					reset := cmd.reset);
				state.alarm.almNC := sys.base.almS(							//NC control only for 4..20 mA
					signal := state.signal < 2.5,
					reset := cmd.reset);
			2: 	//0..10 V
				state.alarm.almSC := sys.base.almS(
					signal := state.signal > 10.5,
					reset := cmd.reset);
			3: 	//-150..+150 C
				state.alarm.almSC := sys.base.almS(
					signal := state.signal > 155.0,
					reset := cmd.reset);
			4: 	//-150..+250 C
				state.alarm.almSC := sys.base.almS(
					signal := state.signal > 255.0,
					reset := cmd.reset);
			ELSE
				state.alarm.almSC := FALSE;
				state.alarm.almNC := FALSE;
		END_CASE
		//ST
		IF state.alarm.almNC OR state.alarm.almSC THEN
			state.alarm.almST := TRUE;
		END_IF
	ELSE
		state.alarm.almSC := FALSE;
		state.alarm.almNC := FALSE;
		state.alarm.almST := FALSE;
	end_if
END_ACTION

ACTION s00_globalCommands:
//global commands
	//emergency signal
		emergency := FALSE;
	//auto mode
		IF sys.allAuto THEN
			CMD.manual := FALSE;
		END_IF;
	//global reset
		IF sys.allreset THEN
			CMD.reset := TRUE;
		END_IF
END_ACTION

ACTION s10_alarms:
//alarms with time control
	//HH
		state.alarm.almHH := sys.base.alm(
			signal := (result > cfg.SP.HH AND cfg.cfg.useHigh),
			reset := (CMD.reset OR NOT CMD.startA) OR (cfg.cfg.useAutoReset AND result <= cfg.SP.HH),
			clock := clock[0].CMD);
	//H
		state.alarm.almH := sys.base.alm(
			signal := (result > cfg.SP.H),
			reset := (CMD.reset OR NOT CMD.startA OR (result < cfg.SP.H)),
			clock := clock[1].CMD);
	//L
		state.alarm.almL := sys.base.alm(
			signal := (result < cfg.SP.L),
			reset := (CMD.reset OR NOT CMD.startA OR (result > cfg.SP.L)),
			clock := clock[2].CMD);
	//LL
		state.alarm.almLL := sys.base.alm(
			signal := (result < cfg.SP.LL AND cfg.cfg.useLow),
			reset := (CMD.reset OR NOT CMD.startA) OR (cfg.cfg.useAutoReset AND result >= cfg.SP.LL),
			clock := clock[3].CMD);
END_ACTION

ACTION s11_reset:
//reset
	IF CMD.reset THEN
		state.state.alarm := FALSE;
		FOR cnt := 0 TO 3 DO
			clock[cnt].CMD.reset := TRUE;
		END_FOR
		CMD.alarm := FALSE;
		CMD.reset := FALSE;
	END_IF
END_ACTION

ACTION s16_timers:
//call timers
	FOR cnt := 0 TO 3 DO
		clock[cnt].SP := INT_TO_REAL(cfg.spT[cnt]) / 10.0;
		sys.timer.rtc (clock[cnt]);
	END_FOR
END_ACTION

ACTION s15_globalData:
//manual mode flag
	IF CMD.manual THEN sys.man.drvAI := TRUE; END_IF;
	
//global alarm
	IF (state.alarm.almST OR state.alarm.almHH OR state.alarm.almLL) AND CMD.startA THEN
		state.state.alarm := TRUE;
		sys.alm.drvAI := TRUE;
		CMD.alarm := TRUE;
	END_IF
END_ACTION

ACTION s02_workMode:
//convert data		
	cmd.startA := cfg.cfg.useEnable;
	//data convert to phisycal value scale
		value := sys.base.conv(
			signal := signal,
			range := cfg.range);
			
	//signal's correction
		IF NOT CMD.startA THEN
			value := 0;
		ELSE
			value := value * cfg.Multiplier + cfg.Calibration;
		END_IF
END_ACTION

ACTION s03_filter:
//signal filter	
	//filtering mode
		Filter(
			start := CMD.startA AND cfg.cfg.useFilter,
			signal := value,
			filterType := cfg.filterType,
			filterLim := cfg.filterLim,
			result => buffer);
			
	//no filtering mode
		IF NOT cfg.cfg.useFilter THEN
			buffer := value;
		END_IF
END_ACTION

ACTION s05_exe:
//device control
	sys.base.exe(emergency := emergency,
		CMD := CMD);
END_ACTION

ACTION s06_delays:

END_ACTION

ACTION s08_turnOFF:

END_ACTION

ACTION s09_options:
//options
	IF cmd.startA THEN
		IF NOT cmd.manual THEN
			state.result := buffer;
		END_IF
	ELSE
		state.result := 0.0;
	END_IF
	
//state signal transfer	
	result := state.result;
END_ACTION

ACTION s12_state:
//state information
	cmd.call := TRUE;
END_ACTION

ACTION s18_netData:
netData.status 	:= state.status;
netData.ap 		:= state.result;
netData.alarm.0 := state.alarm.almST;
netData.alarm.1 := state.alarm.almHH;
//netData.alarm.2 := state.alarm.almH;
//netData.alarm.3 := state.alarm.almL;
netData.alarm.4 := state.alarm.almLL;
netData.alarm.5 := state.alarm.almNC;
netData.alarm.6 := state.alarm.almSC;
END_ACTION

END_FUNCTION_BLOCK

// Drivers/Devices/04. Analog Output/SlowMode/SubFilter
FUNCTION_Block SubFilter
VAR_INPUT
	start			:BOOL;		//Enable filter
	signal			:REAL;		//Input value
	filterType		:INT;		//Execution clock for filter: 0 = every cycle of PLC, 1 = 0.1s, 2 = 1s
	filterLim 		:INT;		//value of records in filter buffer
END_VAR
VAR_OUTPUT
	result			:REAL;		//Median value for all measurments
END_VAR
VAR
	cnt				:INT;		//calculate actual measurments
	x				:INT;		//internal counter for shifting array elements
	exe				:BOOL;		//command to execution filtering cycle
	Summ			:REAL;		//Summary value of all array's values
	DATA			:ARRAY [0..100] OF REAL;
END_VAR

//limit
	IF filterLim > 100 THEN
		filterLim := 100;
	END_IF

//adding new entyty
IF start AND (filterType = 0 OR (filterType = 1 AND sys.pulse01s) OR (filterType = 2 AND sys.pulse1s)) THEN
    IF cnt < filterLim THEN
        cnt := cnt + 1;
    END_IF;
	exe := TRUE;
ELSIF NOT start THEN
	cnt := 0;
	result := signal;
END_IF;

//start cycle
IF exe THEN
	//read new value
	DATA[0] := signal;
	Summ := 0.0;
	
	//limit values
	IF cnt > filterLim THEN
		cnt := filterLim;
	END_IF;
	
	//shifting array
	FOR x := filterLim TO 1 BY -1 DO
		DATA[x] := DATA[x - 1];
		IF x <= cnt AND start THEN
			Summ := Summ + DATA[x];
		END_IF;
	END_FOR;
	
	//calculate median values
	IF cnt > 0 THEN
		result := Summ / cnt;
	ELSE
		result := 0.0;
	END_IF;
	
	//end cycle
	exe := FALSE;
END_IF;

END_FUNCTION_BLOCK

// Drivers/Devices/04. Analog Output/DrvAO
FUNCTION_BLOCK DrvAO
VAR_INPUT
	command			:BOOL;			//Command in automation mode from algorythms
	setPoint		:REAL;			//Control signal from algorythm
END_VAR	
VAR_IN_OUT
	CMD				:udtCMD;		//Non-retain structure with command word
	cfg				:cfgAO;			//Retain structure with settings
	devState		:udtDevAnalog;	
END_VAR
VAR_OUTPUT
	state			:stateAO;		//Non-retain structure with states information
	netData			:udtNetDataAnalog;//Data for network communication via ModBus TCP/RTU
	resultR			:REAL;			//Analog output signal to PLC in REAL
	resultI			:INT;			//Analog output signal to PLC in INT
END_VAR
VAR
	value			:REAL;			//tmp value for calculating 
	buffer			:REAL;			//tnp value for slow mode
	emergency		:BOOL;			//emergency signal
	spA				:REAL;			//setpoint for work
	cnt				:INT;			//internal counter
	PT				:ARRAY [0..1] OF R_TRIG;
	NT				:ARRAY [0..1] OF F_TRIG;
	drvSlow			:subSlow;
END_VAR

//ANALOG OUTPUT
//control of typical analog command
// - Hz setpoint for motors
// - % setpoint for valves

s00_globalCommands();
s01_externalCommand();
//s02_workMode();
//s03_filter();
//s04_alarmsRaw();
s05_exe();
//s06_delays();
//s07_turnON();
//s08_turnOFF();
s09_options();
//s10_alarms();
//s11_reset();
s12_state();
//s13_commands();
//s14_opTime();
s15_globalData();
//s16_timers();
s17_hmi();
s18_netData();
//s19_reserv();
//s20_test();

ACTION s12_state:
//state information
	cmd.call := TRUE;
	//ready
		devState.READY := NOT cmd.lock AND NOT cmd.force AND NOT cmd.alarm AND NOT emergency;
	//busy
		devState.BUSY := cmd.startM AND cfg.spM <> buffer;
	//done
		devState.DONE := cmd.startM AND cfg.spM = buffer;
	//ap
		devState.AP := buffer;
END_ACTION

ACTION s17_hmi:
//hmi data
	//convert data
		state.signal := sys.base.scale(
			value := value,
			inputType := cfg.outputType,
			range := cfg.range);
	//rotate output type
		cfg.outputType := sys.base.inc(
			rotate := cmd.test,
			value := cfg.outputType,
			maxValue := sys.aoMaxValueType);
	//rotate value type
		cfg.valueType := sys.base.inc(
			rotate := cmd.lowSpeed,
			value := cfg.valueType,
			maxValue := sys.aoMaxValueValue);
	//HMI light
		IF cmd.startM AND NOT cmd.alarm THEN state.status := 1; END_IF
		IF NOT cmd.startM AND NOT cmd.alarm THEN state.status := 0; END_IF
		IF cmd.alarm THEN state.status := 5; END_IF 
	//send Status to control structure
		devState.STATUS := state.status;
END_ACTION

ACTION s15_globalData:
//manual mode flag
	IF CMD.manual THEN sys.man.drvAO := TRUE; END_IF;
END_ACTION

ACTION s00_globalCommands:
//global commands
	//emergency signal
		IF cfg.cfg.useNoEmrg THEN
			emergency := FALSE;
		ELSE
			emergency := sys.allBlock;
		END_IF
	//to auto mode
		IF sys.allAuto THEN
			CMD.manual := FALSE;
		END_IF;
	//simulation mode
		PT[0](CLK := sys.allSim);
		NT[0](CLK := sys.allSim);
		IF PT[0].Q THEN cfg.cfg.useSim := TRUE; END_IF;
		IF NT[0].Q THEN cfg.cfg.useSim := FALSE; END_IF;
		IF cfg.cfg.useSim THEN sys.sim.drvAO := TRUE; END_IF;
END_ACTION

ACTION s01_externalCommand:
//select source of control
	IF cfg.cfg.useExt THEN
		CMD.startA := command;
		spA := setPoint;
	ELSE
		CMD.startA := devState.REQ;
		spA := devState.SP;
	END_IF
	IF NOT CMD.manual THEN
		cfg.spM := spA;
	END_IF
END_ACTION

ACTION s05_exe:
//device control
	sys.base.exe(emergency := emergency,
		CMD := CMD);
	//setpoint control
		IF NOT CMD.manual THEN
			cfg.spM := setPoint;
		END_IF
		IF NOT CMD.startM THEN
			cfg.spM := 0;
		END_IF
END_ACTION

ACTION s09_options:
//slow mode for analog output
	drvSlow(
		REQ := cfg.cfg.useSlow,
		signal := cfg.spM,
		cfg := cfg.slowCfg,
		state => state.slowState,
		result => buffer);

//data convert to phisycal value scale
	value := sys.base.conv(
		signal := buffer,
		range := cfg.range);
		
//state signal transfer
	state.result := buffer;
		
//simulation mode
	IF NOT cfg.cfg.useSim THEN
		resultR := value;
		resultI := REAL_TO_INT(value);
	ELSE
		resultR := 0.0;
		resultI := 0;
	END_IF
END_ACTION

ACTION s18_netData:
netData.status 	:= state.status;
netData.ap 		:= state.result;
END_ACTION

END_FUNCTION_BLOCK

// Drivers/Devices/04. Analog Output/SlowMode/SubSlow
FUNCTION_Block SubSlow
VAR_IN_OUT
	REQ				:BOOL;			//Request control
	signal			:REAL;
	cfg				:cfgSlow;
END_VAR
VAR_OUTPUT
	state			:udtState;		//Word of process state
	result			:REAL;
END_VAR
VAR
	reqUp			:BOOL;
	reqDown			:BOOL;
	step			:INT;			//step control for algorythm
	value			:REAL;			//tmp value for calculating 
	delta			:REAL;			//delta between signal and result
	support			:WORD;			//internal command buffer
	cnt				:INT;			//internal counter
	PT				:ARRAY [0..1] OF R_TRIG;
	NT				:ARRAY [0..1] OF F_TRIG;
	clock			:ARRAY [0..2] OF timerRtc;
END_VAR

//Algorithm for slow control analogue value

//global process control
IF NOT cfg.cfg.Enable THEN
	result := signal;
	Step := 0;
END_IF

//algorythm control
	PT[0](CLK := REQ);
	NT[0](CLK := REQ);

//Main process

IF Step = 0 THEN	//wait for start
	IF REQ THEN
		Step := 1;
	ELSIF NT[0].Q THEN
		Step := 20;
	ELSIF NOT REQ THEN
		clock[1].CMD.start := FALSE;
		clock[2].CMD.start := FALSE;
	END_IF
END_IF

IF Step = 1 THEN	//calculate delta
	Delta := signal - result;
	IF Delta > 0 THEN 
		state.Done := FALSE;
		support.0 := FALSE;
		Step := 10;
 	ELSIF Delta < 0 THEN
		state.Done := FALSE;
		support.0 := TRUE;
		Step := 20;
	ELSIF Delta = 0 THEN
		state.Busy := FALSE;
		state.Done := TRUE;
	END_IF;
	Delta := ABS(Delta);	
END_IF

IF Step = 10 THEN	//direction up
	//normal mode
	IF Delta > cfg.spStepUp THEN
		IF cfg.cfg.useUp THEN
			IF value > cfg.spMax THEN
				reqUp := TRUE;
			ELSE
				reqUp := FALSE;
				value := signal;
			END_IF
		ELSE
			reqUp := TRUE;
		END_IF
	ELSE
		reqUp := FALSE;
		value := signal;
	END_IF
	//forced up
	IF PT[0].Q AND cfg.cfg.useForceUp THEN
		reqUp := FALSE;
		value := signal;
	END_IF
	//execute
	IF reqUp THEN
		clock[1].CMD.start := TRUE;
		clock[2].CMD.start := FALSE;
		IF clock[1].CMD.Q THEN
			value := value + cfg.spStepUp;
			clock[1].CMD.start := FALSE;
		END_IF
	END_IF
	//step control finished
	Step := 99;
END_IF



IF Step = 20 THEN	//direction down
	//normal mode
	IF Delta > cfg.spStepDown THEN
		IF cfg.cfg.useUp THEN
			IF value > cfg.spMin THEN
				reqDown := TRUE;
			ELSE
				reqDown := FALSE;
				value := signal;
			END_IF
		ELSE
			reqDown := TRUE;
		END_IF
	ELSE
		reqDown := FALSE;
		value := signal;
	END_IF
	//forced up
	IF NT[0].Q AND cfg.cfg.useForceDown THEN
		value := signal;
	END_IF
	//execute
	IF reqDown THEN
		clock[1].CMD.start := FALSE;
		clock[2].CMD.start := TRUE;
		IF clock[2].CMD.Q THEN
			value := value - cfg.spStepDown;
			clock[2].CMD.start := FALSE;
		END_IF
	END_IF
	//step control finished
	Step := 99;
END_IF


IF Step = 99 THEN	//Finished step
	Step := 0;
END_IF

//call timers
	clock[1].SP := cfg.spTUp;
	clock[2].SP := cfg.spTDown;
	FOR cnt := 0 TO 2 DO
		sys.timer.rtc (clock[cnt]);
	END_FOR

END_FUNCTION_BLOCK

// Drivers/Devices/01. Discrete Input/DrvDI
FUNCTION_Block DrvDI
VAR_INPUT
	signal			:BOOL;		//Physical input value, i.e. %IX0.6
END_VAR
VAR_IN_OUT
	CMD				:udtCMD;	//Non-retain structure with command word
	cfg				:cfgDI;		//Retain structure with settings
END_VAR
VAR_OUTPUT
	netData			:BOOL;		//Data for network communication via ModBus TCP/RTU
	result			:BOOL;		//Logical output value, used in algorythms
END_VAR
VAR
	emergency		:BOOL;		//emergency signal
	value			:BOOL;		//internal signal
	clock			:ARRAY [0..1] OF timerRtc;
END_VAR

//DIGITAL INPUT
//signals from sensors, for example:
//	- keys
//	- sensors
//	- etc

s00_globalCommands();
//s01_externalCommand();
s02_workMode();
s03_filter();
//s04_alarmsRaw();
s05_exe();
//s06_delays();
//s07_turnON();
//s08_turnOFF();
s09_options();
//s10_alarms();
//s11_reset();
s12_state();
//s13_commands();
//s14_opTime();
s15_globalData();
s16_timers();
//s17_hmi();
s18_netData();
//s19_reserv();
//s20_test();

ACTION s00_globalCommands:
//global commands
	//emergency signal
		emergency := FALSE;
	//to auto mode
		IF sys.allAuto THEN
			CMD.manual := FALSE;
		END_IF;
END_ACTION

ACTION s12_state:
//state information
	cmd.call := TRUE;
END_ACTION

ACTION s02_workMode:
//normal close mode
	IF cfg.cfg.useNC THEN
		value := NOT signal;
	ELSE
		value := signal;
	END_IF;
END_ACTION

ACTION s03_filter:
//signal filter	
	IF cfg.cfg.useFilter THEN
	//turn on
		IF cfg.spTOn > 0 AND value THEN
			clock[0].CMD.start := TRUE;
			clock[1].CMD.start := FALSE;
			IF clock[0].CMD.Q THEN
				CMD.startA := value;
			END_IF;
		ELSIF value THEN
			CMD.startA := TRUE;
			clock[0].CMD.start := FALSE;
			clock[1].CMD.start := FALSE;
		END_IF;
			
	//turn off
		IF cfg.spTOff > 0 AND NOT value THEN
			clock[0].CMD.start := FALSE;
			clock[1].CMD.start := TRUE;
			IF clock[1].CMD.Q THEN
				CMD.startA := signal;
			END_IF;
		ELSIF NOT value THEN
			CMD.startA := FALSE;
			clock[0].CMD.start := FALSE;
			clock[1].CMD.start := FALSE;
		END_IF;
	ELSE
		CMD.startA := value;
	END_IF
END_ACTION

ACTION s05_exe:
//device control
	sys.base.exe(emergency := emergency,
		CMD := CMD);
END_ACTION

ACTION s16_timers:
//call timers
	clock[0].SP := cfg.spTOn;
	clock[1].SP := cfg.spTOff;
	sys.timer.rtc (clock[0]);
	sys.timer.rtc (clock[1]);
END_ACTION

ACTION s15_globalData:
//manual mode flag
	IF CMD.manual THEN sys.man.drvDI := TRUE; END_IF;
END_ACTION

ACTION s09_options:
//result
	result := CMD.startM;
END_ACTION

ACTION s18_netData:
netData := result;
END_ACTION

END_FUNCTION_BLOCK

// Drivers/Devices/02. Discrete Output/DrvDO
FUNCTION_Block DrvDO
VAR_INPUT
	command			:BOOL;			//Command in automation mode from algorythms
END_VAR
VAR_IN_OUT
	CMD				:udtCMD;		//Non-retain structure with command word
	cfg				:cfgDO;			//Retain structure with settings	
END_VAR
VAR_OUTPUT
	netData			:BOOL;		//Data for network communication via ModBus TCP/RTU	
	result			:BOOL;			//Phisical output signal, i.e. %QX2.4
END_VAR
VAR
	emergency		:BOOL;			//emergency signal
	PT				:ARRAY [0..1] OF R_TRIG;
	NT				:ARRAY [0..1] OF F_TRIG;
END_VAR

//DIGITAL OUTPUT
//control of primitive devices, for example
// - solenoid valve
// - signal for data exchange with another device
// - etc

s00_globalCommands();
//s01_externalCommand();
//s02_workMode();
//s03_filter();
//s04_alarmsRaw();
s05_exe();
//s06_delays();
//s07_turnON();
//s08_turnOFF();
s09_options();
//s10_alarms();
//s11_reset();
s12_state();
//s13_commands();
//s14_opTime();
s15_globalData();
//s16_timers();
//s17_hmi();
s18_netData();
//s19_reserv();
//s20_test();

ACTION s12_state:
//state information
	cmd.call := TRUE;
END_ACTION

ACTION s15_globalData:
//manual mode flag
	IF CMD.manual THEN sys.man.drvDO := TRUE; END_IF;
END_ACTION

ACTION s00_globalCommands:
//global commands
	//emergency signal
		IF cfg.cfg.useNoEmrg THEN
			emergency := FALSE;
		ELSE
			emergency := sys.allBlock;
		END_IF
	//to auto mode
		IF sys.allAuto THEN
			CMD.manual := FALSE;
		END_IF;
	//simulation mode
		PT[0](CLK := sys.allSim);
		NT[0](CLK := sys.allSim);
		IF PT[0].Q THEN cfg.cfg.useSim := TRUE; END_IF;
		IF NT[0].Q THEN cfg.cfg.useSim := FALSE; END_IF;
		IF cfg.cfg.useSim THEN sys.sim.drvDO := TRUE; END_IF;
END_ACTION

ACTION s05_exe:
//device control
	sys.base.exe(emergency := emergency,
		CMD := CMD);
END_ACTION

ACTION s09_options:
//conditions for turn on and turn off
	IF cmd.startM THEN
		IF cfg.cfg.useNC THEN
			result := NOT cmd.startM;
		ELSE
			result := cmd.startM;
		END_IF
	END_IF
	
//simulation mode
	IF cfg.cfg.useSim THEN
		result := FALSE;
	END_IF;
END_ACTION

ACTION s18_netData:
netData := cmd.startM;
END_ACTION

END_FUNCTION_BLOCK

// Drivers/Devices/05. Motor Direct/DrvM
FUNCTION_Block DrvM
VAR_INPUT
	command			:BOOL;			//Command in automation mode from algorythms
	fbQF			:BOOL;			//Physical input value, control feedback signal 'Ready' or NOT 'alarm'
	fbKM			:BOOL;			//Physical input value, control feedback signal 'In Work' OR 'Run'
END_VAR
VAR_IN_OUT
	CMD				:udtCMD;		//Non-retain structure with command word
	cfg				:cfgM;			//Retain structure with settings
	devState		:udtDevDiscrete;	
END_VAR
VAR_OUTPUT
	state			:stateM;		//Non-retain structure with states information
	netData			:udtNetDataDiscrete;//Data for network communication via ModBus TCP/RTU
	cmdFW			:BOOL;			//Phisical output signal for start device, i.e. %QX2.4
END_VAR
VAR
	emergency		:BOOL;			//emergency signal
	req				:BOOL;			//request for start device
	cnt				:INT;			//internal counter
	step			:INT;			//steps for test
	alm				:ARRAY [0..3] OF BOOL;			//support word for transfer alarms
	PT				:ARRAY [0..1] OF R_TRIG;
	NT				:ARRAY [0..1] OF F_TRIG;
	clock			:ARRAY [0..4] OF timerSec;
END_VAR

//MOTORS
//control of typical motors
// - ventitalitons
// - pumps
// - conveyors
// - etc

s00_globalCommands();
s01_externalCommand();
//s02_workMode();
//s03_filter();
s04_alarmsRaw();
s05_exe();
s06_delays();
s07_turnON();
s08_turnOFF();
s09_options();
s10_alarms();
s11_reset();
s12_state();
//s13_commands();
s14_opTime();
s15_globalData();
s16_timers();
s17_hmi();
s18_netData();
//s19_reserv();
s20_test();

ACTION s16_timers:
//call timers
	clock[0].SP := cfg.spTDelayOn;
	clock[1].SP := cfg.spTDelayOff;
	clock[2].SP := cfg.spTOn;
	clock[3].SP := cfg.spTOff;
	clock[4].SP := cfg.spTest;
	FOR cnt := 0 TO 4 DO
		sys.timer.sec (clock[cnt]);
	END_FOR
END_ACTION

ACTION s15_globalData:
//manual mode flag
	IF CMD.manual THEN sys.man.drvM := TRUE; END_IF;

//global alarm
	IF (state.alarm.almES OR
		state.alarm.almExt OR
		state.alarm.almLink OR
		state.alarm.almQF OR
		state.alarm.almSF OR
		state.alarm.almStart OR
		state.alarm.almStop OR
		state.alarm.almTS) AND NOT cfg.cfg.useSim THEN
		state.state.alarm := TRUE;
		sys.alm.drvM := TRUE;
		CMD.alarm := TRUE;
	END_IF
END_ACTION

ACTION s12_state:
//state information
	cmd.call := TRUE;
	//ready
		devState.READY := NOT cmd.lock AND NOT cmd.force AND NOT cmd.alarm AND NOT cmd.service AND NOT cmd.local AND NOT emergency AND state.status < 4;
	//busy
		devState.BUSY := state.status = 2 OR state.status = 3;
	//done
		devState.DONE := (cmd.startM or cmd.local) AND state.status = 1;

//global commands
	state.signalQF := fbQF;
	state.signalKM := fbKM;
END_ACTION

ACTION s00_globalCommands:
//global commands
	//emergency signal
		IF cfg.cfg.useNoEmrg THEN
			emergency := FALSE;
		ELSE
			emergency := sys.allBlock;
		END_IF
	//to auto mode
		IF sys.allAuto THEN
			CMD.manual := FALSE;
		END_IF;
	//global reset
		IF sys.allreset THEN
			CMD.reset := TRUE;
		END_IF
	//simulation mode
		PT[0](CLK := sys.allSim);
		NT[0](CLK := sys.allSim);
		IF PT[0].Q THEN cfg.cfg.useSim := TRUE; END_IF;
		IF NT[0].Q THEN cfg.cfg.useSim := FALSE; END_IF;
		IF cfg.cfg.useSim THEN sys.sim.drvDOA := TRUE; END_IF;
END_ACTION

ACTION s06_delays:
//delay turn on
	IF cfg.spTDelayOn > 0 AND NOT CMD.manual THEN
		IF CMD.startM THEN
			clock[0].CMD.start := TRUE;
			clock[1].CMD.start := FALSE;
			IF clock[0].CMD.Q THEN
				req := TRUE;
			END_IF
		ELSE
			clock[0].CMD.start := FALSE;
		END_IF
	ELSE
		req := CMD.startM;
	END_IF

//delay turn off
	IF cfg.spTDelayOff > 0 AND NOT CMD.manual THEN
		IF NOT CMD.startM THEN
			clock[1].CMD.start := TRUE;
			clock[0].CMD.start := FALSE;
			IF clock[1].CMD.Q THEN
				req := FALSE;
			END_IF
		ELSE
			clock[1].CMD.start := FALSE;
		END_IF
	ELSE
		req := CMD.startM;
	END_IF
END_ACTION

ACTION s05_exe:
//device control
	sys.base.exe(emergency := emergency,
		CMD := CMD);
END_ACTION

ACTION s01_externalCommand:
//select source of control
	IF cfg.cfg.useExt THEN
		CMD.startA := command;
	ELSE
		CMD.startA := devState.REQ;
	END_IF
END_ACTION

ACTION s09_options:
//simulation mode
	IF cfg.cfg.useSim THEN
		cmdFW := FALSE;
	END_IF
END_ACTION

ACTION s08_turnOFF:
//conditions for turn off
	IF NOT req AND state.status < 4 THEN
		clock[2].CMD.start := FALSE;
		clock[3].CMD.start := TRUE;
		cmdFW := req;
	END_IF
END_ACTION

ACTION s07_turnON:
//conditions for turn on
	IF req AND state.status < 4 THEN
		clock[2].CMD.start := TRUE;
		clock[3].CMD.start := FALSE;
		cmdFW := req;
	END_IF
END_ACTION

ACTION s11_reset:
//reset
	IF CMD.reset THEN
		IF state.status > 4 THEN
			state.status := 0;
		END_IF
		FOR cnt := 0 TO 4 DO
			clock[cnt].CMD.reset := TRUE;
		END_FOR
		state.state.alarm := FALSE;
		state.alarm.almES := FALSE;
		state.alarm.almExt := FALSE;
		state.alarm.almLink := FALSE;
		state.alarm.almSF := FALSE;
		state.alarm.almTS := FALSE;
		CMD.alarm := FALSE;
		CMD.reset := FALSE;
	END_IF
END_ACTION

ACTION s04_alarmsRaw:
//alarms raw
	//emergency stop
		state.alarm.almES := sys.base.almS(
				signal := emergency,
				reset := cmd.reset);
	//QF control
		state.alarm.almQF := sys.base.almS(
				signal := not fbQF,
				reset := cmd.reset OR NOT cfg.cfg.useQF OR cfg.cfg.useSim);
END_ACTION

ACTION s10_alarms:
//alarms with time control
	//start alarm control
		state.alarm.almStart := sys.base.alm(
			signal := (req AND NOT fbKM) AND cfg.cfg.useKM,
			reset := (CMD.reset OR cfg.cfg.useSim OR cmd.local),
			clock := clock[2].CMD);
	//stop alarm control
		state.alarm.almStop := sys.base.alm(
			signal := (NOT req AND fbKM) AND cfg.cfg.useKM,
			reset := (CMD.reset OR cfg.cfg.useSim OR cmd.local),
			clock := clock[3].CMD);
END_ACTION

ACTION s17_hmi:
//hmi data
	//calculate status
		//0 - stop/stopping
			IF NOT cmd.startM AND NOT cmd.alarm THEN
				IF NOT fbKM OR NOT cfg.cfg.useKM THEN
					//stopped succesfully
					state.status := 0;
				ELSE
					//stopping in process
					state.status := 2;
				END_IF
			END_IF
		//1 - start/starting
			IF cmd.startM AND NOT cmd.alarm THEN
				IF fbKM OR NOT cfg.cfg.useKM THEN
					//start succesfully
					state.status := 1;
				ELSE
					//starting in process
					state.status := 3;
				END_IF
			END_IF
		//4 - service
			IF cmd.service THEN
				state.status := 4;
			END_IF
		//5 - alarm QF
			IF state.alarm.almQF THEN
				state.status := 5;
			END_IF
		//6 - alarm while starting
			IF state.alarm.almStart THEN
				state.status := 6;
			END_IF
		//7 - alarm while stopping
			IF state.alarm.almStop THEN
				state.status := 7;
			END_IF
		//8 - no connection
			IF state.alarm.almLink THEN
				state.status := 8;
			END_IF
		//9 - other alarms
			IF state.alarm.almES OR 
				state.alarm.almExt OR 
				state.alarm.almSF OR 
				state.alarm.almLink OR
				state.alarm.almTS THEN
				state.status := 9;
			END_IF
	//simulation mode
		IF cfg.cfg.useSim THEN
			IF cmd.startM THEN
				//start
				state.status := 1;
			ELSE
				//stop
				state.status := 0;
			END_IF
		END_IF
	//send Status to control structure
		devState.STATUS := state.status;
END_ACTION

ACTION s14_opTime:
//control operation time
	sys.base.ot(
		enable 		:= cfg.cfg.useOT,
		devBusy		:= cmdFW,
		reset 		:= CMD.resetOT,
		warning 	:= state.state.warningOT,
		opTime 		:= cfg.opTime,
		opTimeLimit := cfg.opTimeLimit);
END_ACTION

ACTION s20_test:
//test
	IF cmd.test THEN
		CASE step OF
			0:	//reset alarms
				IF cmd.alarm THEN
					cmd.reset := TRUE;
				ELSE
					step := 1;
				END_IF
			1:	//switch to manual mode
				cmd.manual := TRUE;
				cmd.startM := TRUE;
				clock[4].CMD.start := TRUE;
				step := 2;
			2:	//control time
				IF clock[4].cmd.Q THEN
					cmd.startM := FALSE;
					cmd.test := FALSE;
				END_IF
		END_CASE
	ELSE
		clock[4].CMD.start := FALSE;
		step := 0;
	END_IF
END_ACTION

ACTION s18_netData:
netData.status 		:= state.status;
netData.alarm.0		:= state.alarm.almQF;
netData.alarm.1		:= state.alarm.almStart;
netData.alarm.2		:= state.alarm.almStop;
netData.alarm.3		:= state.alarm.almTS;
netData.alarm.4		:= state.alarm.almSF;
netData.alarm.5		:= state.alarm.almExt;
netData.alarm.7		:= state.alarm.almLink;
netData.alarm.8		:= state.alarm.almES;
END_ACTION

END_FUNCTION_BLOCK

// Drivers/Devices/02. Discrete Output/DrvDOA
FUNCTION_Block DrvDOA
VAR_INPUT
	command			:BOOL;			//Command in automation mode from algorythms
	setPoint		:REAL;			//Control signal from algorythm
END_VAR
VAR_IN_OUT
	CMD				:udtCMD;		//Non-retain structure with command word
	cfg				:cfgDOA;		//Retain structure with settings
	devState		:udtDevAnalog;	
END_VAR
VAR_OUTPUT
	result			:BOOL;			//Phisical output signal, i.e. %QX2.4
END_VAR
VAR
	emergency		:BOOL;			//emergency signal
	req				:BOOL;			//request for start device
	busy			:BOOL;
	spA				:REAL;			//setpoint for work
	cnt				:INT;			//internal counter
	PT				:ARRAY [0..1] OF R_TRIG;
	NT				:ARRAY [0..1] OF F_TRIG;
	clock			:ARRAY [0..1] OF timerRtc;
END_VAR

//DIGITAL OUTPUT
//control of primitive devices, for example
// - solenoid valve
// - signal for data exchange with another device
// - etc

s00_globalCommands();
s01_externalCommand();
//s02_workMode();
//s03_filter();
//s04_alarmsRaw();
s05_exe();
//s06_delays();
s07_turnON();
s08_turnOFF();
s09_options();
//s10_alarms();
//s11_reset();
s12_state();
//s13_commands();
//s14_opTime();
s15_globalData();
s16_timers();
//s17_hmi();
//s18_reserv();
//s19_reserv();
//s20_test();

ACTION s12_state:
//state information
	cmd.call := TRUE;
	//ready
		devState.READY := NOT cmd.lock AND NOT cmd.force AND NOT cmd.alarm AND NOT emergency;
	//done
		devState.DONE := cmd.startM;
END_ACTION

ACTION s00_globalCommands:
//global commands
	//emergency signal
		IF cfg.cfg.useNoEmrg THEN
			emergency := FALSE;
		ELSE
			emergency := sys.allBlock;
		END_IF
	//to auto mode
		IF sys.allAuto THEN
			CMD.manual := FALSE;
		END_IF;
	//simulation mode
		PT[0](CLK := sys.allSim);
		NT[0](CLK := sys.allSim);
		IF PT[0].Q THEN cfg.cfg.useSim := TRUE; END_IF;
		IF NT[0].Q THEN cfg.cfg.useSim := FALSE; END_IF;
		IF cfg.cfg.useSim THEN sys.sim.drvDOA := TRUE; END_IF;
END_ACTION

ACTION s01_externalCommand:
//select source of control
	IF cfg.cfg.useExt THEN
		CMD.startA := command;
		spA := setPoint;
	ELSE
		CMD.startA := devState.REQ;
		spA := devState.SP;
	END_IF
	IF NOT CMD.manual THEN
		cfg.spM := spA;
	END_IF
END_ACTION

ACTION s05_exe:
//device control
	sys.base.exe(emergency := emergency,
		CMD := CMD);
END_ACTION

ACTION s06_delays:

END_ACTION

ACTION s16_timers:
//call timers
	clock[0].SP := cfg.spT;
	clock[1].SP := cfg.spT;
	FOR cnt := 0 TO 1 DO
		sys.timer.rtc (clock[cnt]);
	END_FOR
END_ACTION

ACTION s15_globalData:
//manual mode flag
	IF CMD.manual THEN sys.man.drvDOA := TRUE; END_IF;
END_ACTION

ACTION s07_turnON:
//conditions for turn on
	IF cmd.startM THEN
		IF cfg.cfg.usePWM THEN
			IF clock[0].Percent < cfg.spM OR clock[0].Percent < cfg.spMin THEN
				req := TRUE;
			END_IF
		ELSIF cfg.cfg.useImpulse THEN
			IF clock[0].CMD.start AND NOT clock[0].CMD.Q THEN
				req := TRUE;
			ELSE
				req := FALSE;
			END_IF
		ELSE
			req := cmd.startM;
		END_IF
	END_IF
END_ACTION

ACTION s08_turnOFF:
//conditions for turn off
		IF cfg.cfg.usePWM THEN
			IF clock[0].Percent >= cfg.spM OR clock[0].Percent > cfg.spMax THEN
				req := FALSE;
			END_IF
		ELSIF cfg.cfg.useImpulse THEN
			IF clock[0].CMD.start AND NOT clock[0].CMD.Q THEN
				req := TRUE;
			ELSE
				req := FALSE;
			END_IF
		ELSE
			req := cmd.startM;
		END_IF
END_ACTION

ACTION s09_options:
//timer control
	PT[0](CLK := busy AND NOT clock[0].CMD.start);
	NT[0](CLK := busy AND NOT clock[0].CMD.start);
	IF cfg.cfg.usePWM THEN
		clock[0].CMD.start := cmd.startM;
		IF clock[0].CMD.Q THEN
			clock[0].CMD.reset := TRUE;
		END_IF
	ELSIF cfg.cfg.useImpulse THEN
		IF NOT clock[0].CMD.start THEN
			IF cmd.startM THEN
				busy := TRUE;
			ELSE
				busy := FALSE;
			END_IF
		END_IF
		IF PT[0].Q OR NT[0].Q THEN
			clock[0].CMD.start := TRUE;
		END_IF
		IF clock[0].CMD.Q THEN
			clock[1].CMD.start := TRUE;
			IF clock[1].cmd.Q THEN
				clock[0].CMD.start := FALSE;
				clock[1].CMD.start := FALSE;
			END_IF
		END_IF
	ELSE
		clock[0].CMD.start := FALSE;
	END_IF
	
//conditions for turn on and turn off
	IF NOT cfg.cfg.useImpulse THEN
		IF cmd.startM THEN
			IF cfg.cfg.useNC THEN
				result := NOT req;
			ELSE
				result := req;
			END_IF
		END_IF
	ELSE
		result := req;
	END_IF

//simulation mode
	IF cfg.cfg.useSim THEN
		result := FALSE;
	END_IF;
END_ACTION

END_FUNCTION_BLOCK

// Drivers/Devices/06. Valve Discrete/DrvV
FUNCTION_Block DrvV
VAR_INPUT
	command			:BOOL;			//Command in automation mode from algorythms
	fbQF			:BOOL;			//Physical input value, control feedback signal 'Ready' or NOT 'alarm'
	fbOpen			:BOOL;			//Physical input value, control feedback signal 'Open'
	fbClose			:BOOL;			//Physical input value, control feedback signal 'Close'
END_VAR
VAR_IN_OUT
	CMD				:udtCMD;		//Non-retain structure with command word
	cfg				:cfgV;			//Retain structure with settings
	devState		:udtDevDiscrete;	
END_VAR
VAR_OUTPUT
	state			:stateV;		//Non-retain structure with states information
	netData			:udtNetDataDiscrete;//Data for network communication via ModBus TCP/RTU
	cmdOpen			:BOOL;			//Phisical output signal for opening, i.e. %QX2.4
	cmdClose		:BOOL;			//Phisical output signal for closing, i.e. %QX2.5
END_VAR
VAR
	emergency		:BOOL;			//emergency signal
	reqOpen			:BOOL;			//request for open
	reqClose		:BOOL;			//request for close
	cnt				:INT;			//internal counter
	step			:INT;			//steps for test
	alm				:ARRAY [0..3] OF BOOL;			//support word for transfer alarms
	PT				:ARRAY [0..3] OF R_TRIG;
	NT				:ARRAY [0..1] OF F_TRIG;
	clock			:ARRAY [0..4] OF timerSec;
END_VAR

//VALVES
//control of typical air and electrical valves
// - doors
// - dampers
// - valves
// - etc

s00_globalCommands();
s01_externalCommand();
//s02_workMode();
//s03_filter();
s04_alarmsRaw();
s05_exe();
s06_delays();
s07_turnON();
s08_turnOFF();
s09_options();
s10_alarms();
s11_reset();
s12_state();
//s13_commands();
s14_opTime();
s15_globalData();
s16_timers();
s17_hmi();
s18_netData();
//s19_reserv();
s20_test();

ACTION s00_globalCommands:
//global commands
	//emergency signal
		IF cfg.cfg.useNoEmrg THEN
			emergency := FALSE;
		ELSE
			emergency := sys.allBlock;
		END_IF
	//to auto mode
		IF sys.allAuto THEN
			CMD.manual := FALSE;
		END_IF;
	//global reset
		IF sys.allreset THEN
			CMD.reset := TRUE;
		END_IF
	//simulation mode
		PT[0](CLK := sys.allSim);
		NT[0](CLK := sys.allSim);
		IF PT[0].Q THEN cfg.cfg.useSim := TRUE; END_IF;
		IF NT[0].Q THEN cfg.cfg.useSim := FALSE; END_IF;
		IF cfg.cfg.useSim THEN sys.sim.drvDOA := TRUE; END_IF;
END_ACTION

ACTION s01_externalCommand:
//select source of control
	IF cfg.cfg.useExt THEN
		CMD.startA := command;
	ELSE
		CMD.startA := devState.REQ;
	END_IF
END_ACTION

ACTION s04_alarmsRaw:
//alarms raw
	//emergency stop
		state.alarm.almES := sys.base.almS(
				signal := emergency,
				reset := cmd.reset);
	//QF control
		state.alarm.almQF := sys.base.almS(
				signal := fbQF,
				reset := cmd.reset OR NOT cfg.cfg.useQF OR cfg.cfg.useSim);
END_ACTION

ACTION s05_exe:
//device control
	sys.base.exe(emergency := emergency,
		CMD := CMD);
END_ACTION

ACTION s06_delays:
//delay turn on
	IF cfg.spTDelayOn > 0 AND NOT CMD.manual THEN
		IF CMD.startM THEN
			clock[0].CMD.start := TRUE;
			clock[1].CMD.start := FALSE;
			IF clock[0].CMD.Q THEN
				reqOpen := TRUE;
				reqClose := FALSE;
			END_IF
		ELSE
			clock[0].CMD.start := FALSE;
		END_IF
	ELSE
		reqOpen := TRUE;
		reqClose := FALSE;
	END_IF

//delay turn off
	IF cfg.spTDelayOff > 0 AND NOT CMD.manual THEN
		IF NOT CMD.startM THEN
			clock[1].CMD.start := TRUE;
			clock[0].CMD.start := FALSE;
			IF clock[1].CMD.Q THEN
				reqOpen := FALSE;
				reqClose := TRUE;
			END_IF
		ELSE
			clock[1].CMD.start := FALSE;
		END_IF
	ELSE
		reqOpen := FALSE;
		reqClose := TRUE;
	END_IF
END_ACTION

ACTION s07_turnON:
//conditions for open
	IF reqOpen AND state.status < 4 THEN
		clock[2].CMD.start := TRUE;
		clock[3].CMD.start := FALSE;
		cmdOpen := TRUE;
		cmdClose := FALSE;
		IF NOT cfg.cfg.useOnce AND NOT fbOpen THEN
			state.state.posOk := FALSE;
		END_IF
	END_IF
END_ACTION

ACTION s08_turnOFF:
//conditions for turn off
	IF (reqClose AND state.status < 4) OR (cfg.cfg.useCWF AND state.status > 4) THEN
		clock[2].CMD.start := FALSE;
		clock[3].CMD.start := TRUE;
		IF NOT cfg.cfg.useDuo THEN
				cmdOpen := FALSE;
				cmdClose := TRUE;
			ELSE
				cmdOpen := TRUE;
				cmdClose := TRUE;
			END_IF
		IF NOT cfg.cfg.useOnce AND NOT fbClose THEN
			state.state.posOk := FALSE;
		END_IF
	END_IF
END_ACTION

ACTION s09_options:
//electric mode with stop while reach open/close position
	IF NOT cfg.cfg.useAir THEN
		IF reqOpen AND fbOpen THEN
			cmdOpen := FALSE;
			state.state.posOk := TRUE;
		END_IF
		IF reqClose AND fbClose THEN
			cmdClose := FALSE;
			state.state.posOk := TRUE;
		END_IF
	END_IF

//simulation mode
	IF cfg.cfg.useSim THEN
		cmdOpen := FALSE;
		cmdClose := FALSE;
	END_IF
END_ACTION

ACTION s10_alarms:
//alarms with time control
	//start alarm control
		state.alarm.almOpen := sys.base.alm(
			signal := (reqOpen AND NOT fbOpen) AND cfg.cfg.usefbOpen,
			reset := (CMD.reset OR cfg.cfg.useSim OR cmd.local),
			clock := clock[2].CMD);
	//stop alarm control
		state.alarm.almClose := sys.base.alm(
			signal := (reqClose AND NOT fbClose) AND cfg.cfg.usefbClose,
			reset := (CMD.reset OR cfg.cfg.useSim OR cmd.local),
			clock := clock[3].CMD);
END_ACTION

ACTION s11_reset:
//reset
	IF CMD.reset THEN
		IF state.status > 4 THEN
			state.status := 0;
		END_IF
		FOR cnt := 0 TO 4 DO
			clock[cnt].CMD.reset := TRUE;
		END_FOR
		state.state.alarm := FALSE;
		state.alarm.almES := FALSE;
		state.alarm.almClose := FALSE;
		state.alarm.almDuo := FALSE;
		state.alarm.almExt := FALSE;
		state.alarm.almLink := FALSE;
		state.alarm.almOpen := FALSE;
		state.alarm.almQF := FALSE;
		state.alarm.almTS := FALSE;
		CMD.alarm := FALSE;
		CMD.reset := FALSE;
	END_IF
END_ACTION

ACTION s12_state:
//state information
	cmd.call := TRUE;
	//ready
		devState.READY := NOT cmd.lock AND NOT cmd.force AND NOT cmd.alarm AND NOT cmd.service AND NOT cmd.local AND NOT emergency AND state.status < 4;
	//busy
		devState.BUSY := state.status = 2 OR state.status = 3;
	//done
		devState.DONE := (cmd.startM OR cmd.local) AND state.status = 1;

//global commands
	state.signalQF := fbQF;
	state.signalOpen := fbOpen;
	state.signalClose := fbClose;
END_ACTION

ACTION s14_opTime:
//control operation time
	sys.base.ot(
		enable 		:= cfg.cfg.useOT,
		devBusy		:= reqOpen OR reqClose,
		reset 		:= CMD.resetOT,
		warning 	:= state.state.warningOT,
		opTime 		:= cfg.opTime,
		opTimeLimit := cfg.opTimeLimit);
END_ACTION

ACTION s15_globalData:
//manual mode flag
	IF CMD.manual THEN sys.man.drvV := TRUE; END_IF;

//global alarm
	IF (state.alarm.almES OR
		state.alarm.almExt OR
		state.alarm.almLink OR
		state.alarm.almQF OR
		state.alarm.almDuo OR
		state.alarm.almOpen OR
		state.alarm.almClose OR
		state.alarm.almTS) AND NOT cfg.cfg.useSim THEN
		state.state.alarm := TRUE;
		sys.alm.drvV := TRUE;
		CMD.alarm := TRUE;
	END_IF
END_ACTION

ACTION s16_timers:
//call timers
	clock[0].SP := cfg.spTDelayOn;
	clock[1].SP := cfg.spTDelayOff;
	clock[2].SP := cfg.spTOn;
	clock[3].SP := cfg.spTOff;
	clock[4].SP := cfg.spTest;
	FOR cnt := 0 TO 4 DO
		sys.timer.sec (clock[cnt]);
	END_FOR
END_ACTION

ACTION s17_hmi:
//hmi data
	//calculate status
		//0 - stop/stopping
			IF NOT cmd.startM AND NOT cmd.alarm THEN
				IF NOT fbClose OR NOT cfg.cfg.usefbClose THEN
					//stopped succesfully
					state.status := 0;
				ELSE
					//stopping in process
					state.status := 2;
				END_IF
			END_IF
		//1 - start/starting
			IF cmd.startM AND NOT cmd.alarm THEN
				IF fbOpen OR NOT cfg.cfg.usefbOpen THEN
					//start succesfully
					state.status := 1;
				ELSE
					//starting in process
					state.status := 3;
				END_IF
			END_IF
		//4 - service
			IF cmd.service THEN
				state.status := 4;
			END_IF
		//5 - alarm QF
			IF state.alarm.almQF THEN
				state.status := 5;
			END_IF
		//6 - alarm while starting
			IF state.alarm.almOpen THEN
				state.status := 6;
			END_IF
		//7 - alarm while stopping
			IF state.alarm.almClose THEN
				state.status := 7;
			END_IF
		//8 - no connection
			IF state.alarm.almLink THEN
				state.status := 8;
			END_IF
		//9 - other alarms
			IF state.alarm.almES OR 
				state.alarm.almExt OR 
				state.alarm.almDuo OR
				state.alarm.almLink OR
				state.alarm.almTS THEN
				state.status := 9;
			END_IF
	//simulation mode
		IF cfg.cfg.useSim THEN
			IF cmd.startM THEN
				//start
				state.status := 1;
			ELSE
				//stop
				state.status := 0;
			END_IF
		END_IF
	//send Status to control structure
		devState.STATUS := state.status;
END_ACTION

ACTION s20_test:
//test
	IF cmd.test THEN
		CASE step OF
			0:	//reset alarms
				IF cmd.alarm THEN
					cmd.reset := TRUE;
				ELSE
					step := 1;
				END_IF
			1:	//switch to manual mode
				cmd.manual := TRUE;
				cmd.startM := TRUE;
				step := 2;
			2:	//control open
				IF state.status = 1 THEN
					clock[4].CMD.start := TRUE;
					IF clock[4].cmd.Q THEN
						cmd.startM := FALSE;
						step := 3;
					END_IF
				ELSIF state.status > 4 THEN
					step := 4;
				END_IF
			3:	//control close
				IF state.status = 0 OR state.status > 4 THEN
					step := 4;
				END_IF
			4:	//final step
				cmd.test := FALSE;
		END_CASE
	ELSE
		clock[4].CMD.start := FALSE;
		step := 0;
	END_IF
END_ACTION

ACTION s18_netData:
netData.status 		:= state.status;
netData.alarm.0		:= state.alarm.almQF;
netData.alarm.1		:= state.alarm.almOpen;
netData.alarm.2		:= state.alarm.almClose;
netData.alarm.3		:= state.alarm.almTS;
netData.alarm.4		:= state.alarm.almDuo;
netData.alarm.5		:= state.alarm.almExt;
netData.alarm.7		:= state.alarm.almLink;
netData.alarm.8		:= state.alarm.almES;
END_ACTION

END_FUNCTION_BLOCK

// Drivers/Devices/20. PID/DrvPID
FUNCTION_BLOCK DrvPID
VAR_INPUT
	signal			:REAL;			//Analog signal from AI
END_VAR
VAR_IN_OUT
	cmd				:udtCMD;		//Non-retain structure with command word
	cfg				:cfgPID;		//Retain structure with settings
	result			:udtDevAnalog;	//Analog coomand for AO
END_VAR
VAR_OUTPUT
	state			:statePID;		//Non-retain structure with states information
END_VAR
VAR
	value			:REAL;			//tmp value for calculating 
	valueDB			:REAL;
	buffer			:REAL;			//tnp value for slow mode
	resultR			:REAL;
	support			:WORD;			//internal command buffer
	emergency		:BOOL;			//emergency signal
	cnt				:INT;			//internal counter
	range			:listRange;
	alm				:ARRAY [0..3] OF BOOL;			//support word for transfer alarms
	PT				:ARRAY [0..1] OF R_TRIG;
	NT				:ARRAY [0..1] OF F_TRIG;
	clock			:ARRAY [0..3] OF timerRtc;
	PID				:PID;
	maxValueValueIn	:INT := 10;
	maxValueValueOut:INT := 5;
END_VAR

//PID
//control of analog processes

s00_globalCommands();
//s01_externalCommand();
//s02_workMode();
s03_filter();
//s04_alarmsRaw();
s05_exe();
//s06_delays();
s07_turnON();
//s08_turnOFF();
s09_options();
//s10_alarms();
s11_reset();
s12_state();
s13_commands();
//s14_opTime();
s15_globalData();
//s16_timers();
s17_hmi();
//s18_reserv();
//s19_reserv();
//s20_test();

ACTION s07_turnON:
//call PID
	PID(
		ACTUAL 		:= valueDB,
		SET_POINT 	:= cfg.spM,
		KP 			:= cfg.spKP,
		TN 			:= cfg.spTi,
		TV 			:= cfg.spTd,
		Y_MANUAL 	:= cfg.spResult,
		Y_OFFSET 	:= cfg.calibrationIn,
		Y_MIN 		:= range.minIn,
		Y_MAX 		:= range.maxIn,
		MANUAL 		:= CMD.service,
		RESET 		:= CMD.reset,
		Y 			=> buffer,
		LIMITS_ACTIVE => state.alarm.almLimits,
		OVERFLOW	  => state.alarm.almOveFlow);
		
//control PID
	IF CMD.startM OR CMD.service THEN
		CMD.reset := FALSE;
	ELSE
		CMD.reset := TRUE;
		buffer := 0.0;
	END_IF
END_ACTION

ACTION s06_delays:

END_ACTION

ACTION s05_exe:
//device control
 	sys.base.exe(emergency := emergency,
 			CMD := CMD);
	//manual mode flag
		IF CMD.manual THEN 
			sys.man.drvPID := TRUE;
		ELSE
			cfg.spM := cfg.spA; 
		END_IF;
		IF NOT CMD.service THEN
			cfg.spResult := buffer;
		END_IF
END_ACTION

ACTION s03_filter:
//convert data
	state.signalPID := signal;
	//data input scaling 0-100
		IF cfg.cfg.useScaleIn THEN
			cfg.rangeIn.minOut := 0;
			cfg.rangeIn.maxOut := 100;
			value := sys.base.conv(
				signal := signal,
				range := cfg.rangeIn);
			value := value * cfg.multiplierIn;
			range.minIn := cfg.rangeIn.minIn;
			range.maxIn := cfg.rangeIn.maxIn;
			cfg.cfg.useCorrectionIn := FALSE;
		END_IF
	//data converting
		IF cfg.cfg.useCorrectionIn THEN
			value := value * cfg.multiplierIn + cfg.calibrationIn;
			range.minIn := cfg.rangeIn.minIn * cfg.multiplierIn;
			range.maxIn := cfg.rangeIn.maxIn * cfg.multiplierIn;
			cfg.cfg.useScaleIn := FALSE;
		END_IF
	//dead band control
		IF cfg.cfg.useDB THEN
			range.minOut := cfg.spA - cfg.spDB;
			range.maxOut := cfg.spA + cfg.spDB;
			IF value < range.minOut OR value > range.maxOut THEN
				valueDB := value;
			END_IF
		ELSE
			valueDB := value;
		END_IF
END_ACTION

ACTION s00_globalCommands:
//global commands
	//emergency signal
		IF cfg.cfg.useNoEmrg THEN
			emergency := FALSE;
		ELSE
			emergency := sys.allBlock;
		END_IF
//global commands
	state.state.call := TRUE;
	//auto mode
		IF sys.allAuto THEN
			CMD.manual := FALSE;
			CMD.Force := FALSE;
		END_IF;
	//simulation mode
		PT[0](CLK := sys.allSim);
		NT[0](CLK := sys.allSim);
		IF PT[0].Q THEN cfg.cfg.useSim := TRUE; END_IF;
		IF NT[0].Q THEN cfg.cfg.useSim := FALSE; END_IF;
		IF cfg.cfg.useSim THEN sys.sim.drvPID := TRUE; END_IF;
END_ACTION

ACTION s09_options:
//convert data
	//data output scaling
		IF cfg.cfg.useScaleOut THEN
			cfg.rangeOut.minIn := 0;
			cfg.rangeOut.maxIn := 100;
			resultR := sys.base.conv(
				signal := buffer,
				range := cfg.rangeOut);
			resultR := resultR * cfg.multiplierOut;
			IF cfg.cfg.useCorrectionOut THEN
				resultR := resultR + cfg.calibrationOut;
			END_IF
		ELSE
			resultR := buffer;
		END_IF
		state.resultPID := resultR;
END_ACTION

ACTION s11_reset:
//reset
	IF CMD.reset THEN
		state.state.alarm := FALSE;
		FOR cnt := 0 TO 3 DO
			clock[cnt].CMD.reset := TRUE;
		END_FOR
		CMD.alarm := FALSE;
		CMD.reset := FALSE;
	END_IF
END_ACTION

ACTION s12_state:
//state information
	cmd.call := TRUE;
END_ACTION

ACTION s15_globalData:
//manual mode flag
	IF CMD.manual THEN sys.man.drvPID := TRUE; END_IF;
END_ACTION

ACTION s17_hmi:
	//rotate value type
		cfg.typeInput := sys.base.inc(
			rotate := cmd.lowSpeed,
			value := cfg.typeInput,
			maxValue := maxValueValueIn);
	//rotate value type
		cfg.typeOutput := sys.base.inc(
			rotate := cmd.resetOT,
			value := cfg.typeOutput,
			maxValue := maxValueValueOut);
END_ACTION

ACTION s13_commands:
result.SP := resultR;
result.REQ := cmd.startM;
END_ACTION

END_FUNCTION_BLOCK

// Drivers/Devices/10. Flowmeter/DrvFlow
FUNCTION_Block DrvFlow
VAR_INPUT
	signalDI		:BOOL;			//Discrete impulse from flowmeter
	signalAI		:REAL;			//Analog data from flowmeter
END_VAR	
VAR_IN_OUT
	CMD				:udtCMD;		//Non-retain structure with command word
	cfg				:cfgFlow;		//Retain structure with settings
END_VAR
VAR_OUTPUT
	state			:stateFlow;		//Non-retain structure with states information
	netData			:udtNetDataAnalog;//Data for network communication via ModBus TCP/RTU
	PreDone			:BOOL;			//PreSP reached
	Done			:BOOL;			//SP reached
	result			:REAL;			//signal from flowmeter
END_VAR
VAR
	AP				:REAL;			//Actual time for countimng
	AP_POU			:REAL;			//Last actual value for counting
	SW				:REAL;			//start weight for control 
	value			:REAL;			//tmp value for calculating 
	support			:WORD;			//internal command buffer
	emergency		:BOOL;			//emergency signal
	cnt				:INT;			//internal counter
	PT				:ARRAY [0..1] OF R_TRIG;
	NT				:ARRAY [0..1] OF F_TRIG;
	clock			:ARRAY [0..1] OF timerRtc;
	Filter			:subFilter;
END_VAR

//FLOWMETER
//control of typical flowmeter control
// - value of source product
// - flowspeed
// - statistics
// - etc

s00_globalCommands();
//s01_externalCommand();
s02_workMode();
s03_filter();
//s04_alarmsRaw();
s05_exe();
//s06_delays();
//s07_turnON();
//s08_turnOFF();
s09_options();
//s10_alarms();
s11_reset();
s12_state();
//s13_commands();
//s14_opTime();
s15_globalData();
s16_timers();
s17_hmi();
s18_netData();
//s19_reserv();
//s20_test();

ACTION s00_globalCommands:
//global commands
	//global commands
	state.state.call := TRUE;
	//auto mode
		IF sys.allAuto THEN
			CMD.manual := FALSE;
		END_IF;
	//global reset
		IF sys.allreset THEN
			CMD.reset := TRUE;
		END_IF
END_ACTION

ACTION s05_exe:
//device control
	sys.base.exe(emergency := emergency,
				CMD := CMD);
	//reset counter
		PT[1](CLK := CMD.startM);
		IF PT[1].Q THEN
			state.lastAp := state.AP;
			state.AP := 0.0;
		END_IF
END_ACTION

ACTION s09_options:
//summary flow control
	IF CMD.startM THEN
		//flow actual calculating
		IF cfg.cfg.useDI THEN
			//for DI
			state.AP := state.AP + cfg.weight;
		ELSIF NOT cfg.cfg.useFM THEN
			//for AI
			IF sys.pulse01s THEN
				CASE cfg.sizeTime OF
					0:	state.AP := state.AP + result / 3600 / 10;
					1:	state.AP := state.AP + result / 60 / 10;
					2:	state.AP := state.AP + result / 10;
				END_CASE 
			END_IF 
		END_IF 
		//pre-setpoint control
		IF state.AP >= cfg.spPre THEN
			state.state.posOk := TRUE;
		END_IF
		//setpoint control
		IF (state.AP >= (cfg.SP - cfg.DB)) THEN
			state.state.Done := TRUE;
		END_IF
	END_IF
END_ACTION

ACTION s11_reset:
//reset
	IF CMD.reset THEN
		state.state.alarm := FALSE;
		CMD.alarm := FALSE;
		CMD.reset := FALSE;
	END_IF
END_ACTION

ACTION s12_state:
//data transfer
	PreDone := state.state.posOk;
	Done := state.state.Done;
//deactivate control
	NT[0](CLK := CMD.startM);
	IF NT[0].Q THEN
		state.state.posOk := FALSE;
		state.state.Done := FALSE;
	END_IF
END_ACTION

ACTION s15_globalData:
//manual mode flag
		IF CMD.manual THEN sys.man.drvFlow := TRUE; END_IF;
END_ACTION

ACTION s16_timers:
//call timers
	FOR cnt := 0 TO 1 DO
		sys.timer.rtc (clock[cnt]);
	END_FOR
END_ACTION

ACTION s17_hmi:
//HMI light
	IF cfg.cfg.useLight THEN
		IF CMD.startM AND NOT state.state.posOk THEN state.status := 3; END_IF
		IF CMD.startM AND state.state.posOk AND NOT state.state.Done THEN state.status := 2; END_IF
		IF state.state.Done THEN state.status := 1; END_IF
		IF NOT CMD.startM THEN state.status := 0; END_IF
	ELSE
		state.status := 0;
	END_IF
END_ACTION

ACTION s02_workMode:
//impulse mode
	PT[0](CLK := signalDI);
	IF cfg.cfg.useDI AND NOT cfg.cfg.useFM THEN
		IF NOT cfg.cfg.usePOU THEN
			//time reset
			IF PT[0].Q THEN
				clock[0].CMD.reset := TRUE;
				AP := clock[0].AP;
			END_IF 
			//time control
			clock[0].CMD.start := CMD.startM;
		ELSE
			IF NOT PT[0].Q THEN
				AP_POU := AP_POU + cfg.clock;
				AP := AP_POU;
			ELSE
				AP_POU := 0;
			END_IF
		END_IF
	ELSE
		clock[0].CMD.start := FALSE;
	END_IF
	
//weight mode
	IF  cfg.cfg.useFM THEN
		IF NOT support.2 AND CMD.startM THEN
			SW := signalAI;
			support.2 := TRUE;
		END_IF
		IF support.2 THEN
			IF NOT cfg.cfg.useFMAdd THEN
				AP := SW - signalAI;
			ELSE
				AP := signalAI - SW;
			END_IF
		END_IF
	END_IF
END_ACTION

ACTION s03_filter:
//signal's filter
	IF cfg.cfg.useDI THEN
		//discrete input filtering
		IF PT[0].Q THEN
			Filter(
				start := CMD.startM,
				signal := AP,
				filterType := 0,
				filterLim := cfg.filterLim,
				result => result);
		END_IF
	ELSE
		//analog input filtering
		Filter(
			start := CMD.startM AND cfg.cfg.useFilter,
			signal := signalAI,
			filterType := cfg.filterType,
			filterLim := cfg.filterLim,
			result => result);
		IF NOT cfg.cfg.useFilter THEN
			result := value;
		END_IF
	END_IF
	
//state signal transfer
	state.result := result;
END_ACTION

ACTION s18_netData:
netData.status 	:= state.status;
netData.ap 		:= state.result;
END_ACTION

END_FUNCTION_BLOCK

// System/pou00_Start
PROGRAM pou00_Start
VAR
	pulse01s			:UDINT;
	pulse1s				:UDINT;
	clock01s			:UDINT;
	clock05s			:UDINT;
	clock1s				:UDINT;
	
	errDTsplit			:ERROR;
	
	PT					:ARRAY [0..1] OF R_TRIG;
	NT					:ARRAY [0..1] OF F_TRIG;
END_VAR

//Write system time
	

//Read system time
	sys.upTime := TIME();
	sys.upTimeMs := TIME_TO_UDINT(sys.UpTime);
	sys.DAT := ULINT_TO_DT(GetDateTime());
	dtl();
	
//Read library version
	sys.LibVersion := GetLibVersion();

//Pulse generation
	pulse();
		
//clock generation
	clock();
	
//retain save and load
	sys.retainControl(
		retainFileName := sys.retainFileName);

ACTION pulse:
	//pulse 100 ms
		IF (sys.upTimeMs - pulse01s) >= 100 THEN
			sys.pulse01s := TRUE;
			pulse01s := sys.upTimeMs;
		else
			sys.pulse01s := FALSE;
		END_IF;
	//pulse 1 s
		IF (sys.upTimeMs - pulse1s) >= 1000 THEN
			sys.pulse1s := TRUE;
			pulse1s := sys.upTimeMs;
		else
			sys.pulse1s := FALSE;
		END_IF;
		
	//pulse 1 minute
		pulseOne(
			ap 		:= sys.DTL.minute, 
			sp 		:= sys.DTLpulse.minute, 
			signal 	=> sys.pulseMinute);
	
	//pulse 1 hour
		pulseOne(
			ap 		:= sys.DTL.hour, 
			sp 		:= sys.DTLpulse.hour, 
			signal 	=> sys.pulseHour);
			
	//pulse 1 day
		pulseOne(
			ap 		:= sys.DTL.day, 
			sp 		:= sys.DTLpulse.day, 
			signal 	=> sys.pulseDay);
			
	//pulse 1 month
		pulseOne(
			ap 		:= sys.DTL.month, 
			sp 		:= sys.DTLpulse.month, 
			signal 	=> sys.pulseMonth);
			
	//pulse 1 year
		pulseOne(
			ap 		:= sys.DTL.year, 
			sp 		:= sys.DTLpulse.year, 
			signal 	=> sys.pulseYear);
END_ACTION

ACTION clock:
//clock 100 ms
		IF (sys.upTimeMs - clock01s) >= 100 THEN
			IF NOT sys.clock01s THEN
				sys.clock01s := TRUE;
			ELSE
				sys.clock01s := FALSE;
			END_IF;
			clock01s := sys.upTimeMs;
		END_IF;
		
	//clock 500 ms
		IF (sys.upTimeMs - clock05s) >= 500 THEN
			IF NOT sys.clock05s THEN
				sys.clock05s := TRUE;
			ELSE
				sys.clock05s := FALSE;
			END_IF;
			clock05s := sys.upTimeMs;
		END_IF;
		
	//clock 1 s
		IF (sys.upTimeMs - clock1s) >= 1000 THEN
			IF NOT sys.clock1s THEN
				sys.clock1s := TRUE;
			ELSE
				sys.clock1s := FALSE;
			END_IF;
			clock1s := sys.upTimeMs;
		END_IF;
END_ACTION

ACTION dtl:
//convert data_and_time to DTL
	//main values
	errDTsplit := SplitDateTime(
		uliDateTime 	:= GetDateTime(),
		uiYear 			=> sys.DTL.year,
		uiMonth 		=> sys.DTL.millisecond,
		uiDay 			=> sys.DTL.day,
		uiHour 			=> sys.DTL.hour,
		uiMinute 		=> sys.DTL.minute,
		uiSecond 		=> sys.DTL.second,
		uiMilliseconds 	=> sys.DTL.millisecond,
		eWeekday 		=> sys.DTL.weekDay);
END_ACTION

METHOD pulseOne
VAR_INPUT
	ap				:UINT;
END_VAR
VAR_IN_OUT
	sp				:UINT;
END_VAR
VAR_OUTPUT
	signal			:BOOL;
END_VAR
END_METHOD

END_PROGRAM

// System/Library Methods/GetLibVersion
// This function has been automatically generated from the project information.
FUNCTION GetLibVersion : VERSION
VAR_INPUT
	
END_VAR

GetLibVersion.uiMajor := 0;
GetLibVersion.uiMinor := 4;
GetLibVersion.uiServicePack := 0;
GetLibVersion.uiPatch := 0;

END_FUNCTION

// Drivers/Devices/06. Valve Discrete/SubCalibration
FUNCTION_Block SubCalibration
VAR_INPUT
	REQ				:BOOL;			//Request control
	Lim_FW			:BOOL;			//Limit switch forward
	Lim_RV			:BOOL;			//Limit switch rewers
	Mode			:BOOL;			//Claibration mode: 0 - RV->RW-RV, 1 - RW->RV-RW
END_VAR
VAR_OUTPUT
	CMD_FW			:BOOL;			//Command to move froward
	CMD_RV			:BOOL;			//Command to move reverse
	SP_FW			:REAL;			//result time for forward moving
	SP_RV			:REAL;			//result time for reverse moving
	state			:udtState;		//Word of process state
END_VAR
VAR
	Step			:INT;			//step control for algorythm
	value			:REAL;			//tmp value for calculating 
	support			:WORD;			//internal command buffer
	cnt				:INT;			//internal counter
	PT				:ARRAY [0..1] OF R_TRIG;
	NT				:ARRAY [0..1] OF F_TRIG;
	clock			:ARRAY [0..2] OF timerCnt;
END_VAR

//Algorithm for calibrating time for movement in two directions using limit switches

//global process control
IF NOT REQ THEN
	Step := 0;
END_IF
		
//Main process
CASE Step OF
	0:	//wait for start
		IF NOT REQ THEN
			CMD_FW := FALSE;
			CMD_RV := FALSE;
			state.Busy := FALSE;
			state.Done := FALSE;
			FOR cnt := 0 TO 2 DO
				clock[cnt].One := 0.1;
				clock[cnt].CMD.start := FALSE;
				clock[cnt].CMD.Pause := FALSE;
			END_FOR
		ELSE
			state.Busy := TRUE;
			Step := 1;
		END_IF
	1:	//moving to start position
		IF NOT Mode THEN
			IF NOT Lim_FW THEN
				CMD_FW := TRUE;
			ELSE
				CMD_FW := FALSE;
				Step := 2;
			END_IF
		ELSE
			IF NOT Lim_RV THEN
				CMD_RV := TRUE;
			ELSE
				CMD_RV := FALSE;
				Step := 2;
			END_IF
		END_IF
	2:	//control time to 1st direction
		IF NOT Mode THEN
			CMD_FW := FALSE;
			CMD_RV := TRUE;
		ELSE
			CMD_FW := TRUE;
			CMD_RV := FALSE;
		END_IF
		clock[1].CMD.start := TRUE;
		IF (Lim_FW AND Mode) OR (Lim_RV AND NOT Mode) THEN
			IF NOT Mode THEN
				SP_RV := clock[1].AP;
			ELSE
				SP_FW := clock[1].AP;
			END_IF
			clock[1].CMD.Pause := TRUE;
			CMD_FW := FALSE;
			CMD_RV := FALSE;
			Step := 3;
		END_IF
	3:	//control time to 2nd direction
		IF NOT Mode THEN
			CMD_FW := TRUE;
			CMD_RV := FALSE;
		ELSE
			CMD_FW := FALSE;
			CMD_RV := TRUE;
		END_IF
		clock[2].CMD.start := TRUE;
		IF (Lim_FW AND NOT Mode) OR (Lim_RV AND Mode) THEN
			IF Mode THEN
				SP_RV := clock[2].AP;
			ELSE
				SP_FW := clock[2].AP;
			END_IF
			clock[2].CMD.Pause := TRUE;
			CMD_FW := FALSE;
			CMD_RV := FALSE;
			Step := 99;
		END_IF
	99:	//Final step
		state.Busy := FALSE;
		state.Done := TRUE;
END_CASE

//Control time move to 1st direction
sys.timer.cnt(
	signal := sys.pulse01s,
	T := clock[1]);
	
//Control time move to 2nd direction
sys.timer.cnt(
	signal := sys.pulse01s,
	T := clock[2]);

END_FUNCTION_BLOCK

// System/Library Methods/DrvBase
FUNCTION_BLOCK DrvBase
VAR_INPUT
END_VAR
VAR_OUTPUT
END_VAR
VAR
END_VAR

METHOD scale : REAL
VAR_INPUT
	value			:REAL;			//Analog input signal from PLC
	inputType		:INT;			//Input type: 0 = 0..20, 1 = 4..20, 2 = 0..10, 3 = Pt100, 4 = Pt1000
	range			:listrange;		//signal scale range
END_VAR
VAR
	typeMin			:REAL;			//Minimum limit
	typeMax			:REAL;			//Maximum limit
END_VAR
//configuration transfering	
CASE inputType OF
	0: typeMin := 0.0; typeMax := 20.0;
	1: typeMin := 4.0; typeMax := 20.0;
	2: typeMin := 0.0; typeMax := 10.0;
	3: scale := value;
	4: scale := value;
END_CASE

//calculate real input value
IF inputType < 3 THEN
	scale := (value / ((range.maxIn - range.minIn) /  (typeMax - typeMin))) + typeMin;
END_IF
END_METHOD

METHOD conv : REAL
VAR_INPUT
	signal			:REAL;			//Analog input signal from PLC
	range			:listrange;	//signal scale range
END_VAR
VAR
	inv				:BOOL;			//inverse range
	rangeIn			:REAL;			//full input range
	rangeOut		:REAL;			//full value range
	RR_Scale		:REAL;			//range in to range out scale
	valueMin		:REAL;			//actual minimum output value
	valueMax		:REAL;			//actual maximum output value
	Buffer			:REAL;			//tmp value for calculating
END_VAR
//Диапазон входного сигнала
IF range.minIn >= 0 THEN
    rangeIn := range.maxIn - range.minIn;
ELSE
    rangeIn := range.maxIn + ABS(range.minIn);
END_IF;

//Диапазон выходного сигнала
inv := FALSE;
IF range.minOut >= 0 AND range.maxOut >= 0 THEN
    IF range.maxOut > range.minOut THEN
        rangeOut := range.maxOut - range.minOut;
        valueMin := range.minOut;
        valueMax := range.maxOut;
    END_IF;
    IF range.maxOut < range.minOut THEN
        rangeOut := range.minOut - range.maxOut;
        valueMin := range.maxOut;
        valueMax := range.minOut;
		inv := TRUE;
    END_IF;
END_IF;
IF range.minOut <= 0 AND range.maxOut >= 0 THEN
    rangeOut := range.maxOut + ABS(range.minOut);
	valueMin := range.minOut;
    valueMax := range.maxOut;
END_IF;
IF range.minOut <= 0 AND range.maxOut <= 0 THEN
    rangeOut := ABS(range.maxOut) + ABS(range.minOut);
	valueMin := range.minOut;
    valueMax := range.maxOut;
END_IF;
IF range.minOut >= 0 AND range.maxOut <= 0 THEN
    rangeOut := ABS(range.maxOut) + ABS(range.minOut);
	valueMin := range.maxOut;
    valueMax := range.minOut;
END_IF;

//Соотношение диапазонов
IF rangeOut <> 0 THEN
	RR_Scale := rangeIn / rangeOut;
END_IF

//Линеаризация
IF RR_Scale <> 0 THEN
	Buffer := signal / RR_Scale;
END_IF

//Коррекция
Buffer := Buffer + valueMin;

//Инверсия
IF inv THEN
    Buffer := valueMax - Buffer;
END_IF;

//Ограничение снизу
IF Buffer < valueMin THEN
    Buffer := valueMin;
END_IF;

//Ограничение сверху
IF Buffer > valueMax THEN
    Buffer := valueMax;
END_IF;

//Вывод значения
conv := Buffer;
END_METHOD

METHOD alm : BOOL
VAR_INPUT
	signal			:BOOL;		//alarm condition
	reset			:BOOL;		//local reset command
END_VAR
VAR_IN_OUT
	clock			:udtTimer;
END_VAR
//Standart alarm control function
	//Conditions compelete
		IF signal THEN
			clock.start := TRUE;
		ELSE
			clock.start := FALSE;
		END_IF
	//alarm control
		IF clock.Q THEN
			alm := TRUE;
		END_IF
	//alarm reset
		IF sys.allReset OR reset THEN
			clock.start := FALSE;
			alm := FALSE;
		END_IF
END_METHOD

METHOD almS : BOOL
VAR_INPUT
	signal			:BOOL;		//alarm condition
	reset			:BOOL;		//local reset command
END_VAR
//Standart alarm control function Small (without timer)
	//Conditions compelete
		IF signal THEN
			almS := TRUE;
		END_IF
	//alarm reset
		IF sys.allReset OR reset THEN
			almS := FALSE;
		END_IF
END_METHOD

METHOD ot : BOOL
VAR_INPUT
	enable			:BOOL;
	devBusy			:BOOL;
END_VAR
VAR_IN_OUT
	reset			:BOOL;
	warning			:BOOL;
	opTime			:REAL;
	opTimeLimit		:REAL;
END_VAR
//calculate operation time for device
IF enable THEN
	//check status
	IF devBusy THEN
		IF sys.pulse1s THEN
			opTime := opTime + sys.second;
		END_IF
	END_IF
	//check warning
	IF opTime >= opTimeLimit THEN
		warning := TRUE;
	END_IF
	//reset operation time
	IF reset THEN
		opTime := 0;
		reset := FALSE;
		warning := FALSE;	
	END_IF
ELSE
	reset := FALSE;
	warning := FALSE;
END_IF
END_METHOD

